Registration_publishes_a_complete_capability();
Duplicate_key_is_refused_and_the_first_stands();
Write_reaches_the_owning_child_through_the_walk();
Stale_revision_is_refused();
Range_type_and_domain_are_enforced();
RequiresReady_follows_the_root_state();
Unknown_key_and_foreign_scope_change_nothing();
Module_invariant_hook_can_refuse();
Units_and_choices_publish_codes_and_labels();

// One-time setup, on the first test to run rather than in a constructor: the
// suite's own Setup return value is itself an assertion below.
METHOD PRIVATE _M_Arm
IF NOT _init THEN
    _init := TRUE;
    _setupOk := _u.Setup(Name := 'Test.CfgUnit');
    _u();
END_IF
END_METHOD

// Walk the real manifest the way a client does — page by page until the key
// appears — so these tests read exactly what the HMI would be given, not an
// internal shortcut into the registry.
METHOD PRIVATE _M_FetchCapability : BOOL
VAR_INPUT
    Key : STRING(160);
END_VAR
VAR
    page  : INT;
    i     : INT;
    pages : INT;
END_VAR
_M_FetchCapability := FALSE;
pages := 1;
FOR page := 0 TO 63 DO
    IF page >= pages THEN
        RETURN;
    END_IF
    _pager.M_Setup(Target := ADR(_page), PageIndex := page, Revision := 1);
    _u.M_AppendConfig(Pager := _pager);
    _pager.M_Finish();
    pages := _page.PageCount;
    FOR i := 1 TO _page.EntryCount DO
        IF _page.Entries[i].WriteKey = Key THEN
            _found := _page.Entries[i];
            _M_FetchCapability := TRUE;
            RETURN;
        END_IF
    END_FOR
END_FOR
END_METHOD

METHOD Registration_publishes_a_complete_capability
TEST('Registration_publishes_a_complete_capability');
_M_Arm();
AssertTrue(Condition := _setupOk,
    Message := 'a registration that fails must fail Setup, not go quiet');
AssertTrue(Condition := _M_FetchCapability(Key := 'probe.settleTime'),
    Message := 'a registered value appears in the root manifest walk');
AssertEquals_STRING(Expected := 'Test.CfgUnit.Child', Actual := _found.Scope,
    Message := 'the capability is scoped to the module that owns it');
AssertTrue(Condition := _found.Writable,
    Message := 'registration is what makes an entry writable (3.10.2)');
AssertEquals_UDINT(Expected := 1, Actual := _found.WriteRevision,
    Message := 'a writable entry carries a non-zero revision');
AssertEquals_DINT(Expected := TO_DINT(E_ConfigValueType.DURATION),
    Actual := TO_DINT(_found.ValueType),
    Message := 'a TIME publishes as DURATION (TC3 3.8)');
AssertEquals_DINT(Expected := TO_DINT(E_ConfigKind.STATION_CFG),
    Actual := TO_DINT(_found.ConfigKind),
    Message := 'deployment data publishes as STATION_CFG');
AssertEquals_STRING(Expected := 'ms', Actual := _found.Unit,
    Message := 'a duration carries its engineering unit');
AssertEquals_STRING(Expected := '500', Actual := _found.ValueText,
    Message := 'the published value is the live target, in whole milliseconds');
AssertTrue(Condition := _found.RequiresReady,
    Message := 'the declared state requirement reaches the client');
AssertEquals_REAL(Expected := 5000.0, Actual := TO_REAL(_found.Maximum),
    Delta := 0.001, Message := 'declared bounds reach the client');
TEST_FINISHED();
END_METHOD

// Core 0.14: a unit is a CODE the HMI translates (the text is derived from it
// for older clients), and a choice names the catalog prefix that labels each of
// its values - so an editor renders a translated dropdown, never a number.
METHOD Units_and_choices_publish_codes_and_labels
TEST('Units_and_choices_publish_codes_and_labels');
_M_Arm();
AssertTrue(Condition := _M_FetchCapability(Key := 'probe.settleTime'),
    Message := 'the duration is published');
AssertEquals_DINT(Expected := TO_DINT(E_EngUnit.MILLISECOND),
    Actual := TO_DINT(_found.UnitCode),
    Message := 'a duration carries the millisecond CODE');
AssertEquals_STRING(Expected := 'ms', Actual := _found.Unit,
    Message := 'and the legacy text is derived from it, not written separately');
AssertTrue(Condition := _M_FetchCapability(Key := 'probe.retries'),
    Message := 'the unitless number is published');
AssertEquals_DINT(Expected := TO_DINT(E_EngUnit.NONE),
    Actual := TO_DINT(_found.UnitCode), Message := 'NONE = no unit');
AssertEquals_STRING(Expected := '', Actual := _found.Unit,
    Message := 'so an HMI shows no unit text');
AssertTrue(Condition := _M_FetchCapability(Key := 'probe.mode'),
    Message := 'the choice is published');
AssertEquals_STRING(Expected := '0|1|2', Actual := _found.EnumDomain,
    Message := 'with its exact accepted values');
AssertEquals_STRING(Expected := 'project.test.modeValue', Actual := _found.EnumLabelKey,
    Message := 'and the catalog prefix that labels each of them');
AssertFalse(Condition := _dup.M_RegisterConfigChoice(Key := 'probe.empty',
    Item := 'StationCfg/Empty', LabelKey := '', Kind := E_ConfigKind.STATION_CFG,
    Storage := E_ConfigStorage.AS_DINT, pTarget := ADR(_dup.Mode), Domain := '',
    EnumLabelKey := '', RequiresReady := FALSE),
    Message := 'a choice with no choices is refused, not accepted as anything');
TEST_FINISHED();
END_METHOD

METHOD Duplicate_key_is_refused_and_the_first_stands
TEST('Duplicate_key_is_refused_and_the_first_stands');
_M_Arm();
AssertTrue(Condition := _dup.Setup(Name := 'Test.CfgDup'),
    Message := 'the probe registers cleanly the first time');
// Re-registering the same key is the §3.10.2 duplicate case. It fails closed,
// which here means the SECOND caller is refused and the first target stays bound
// — nothing can tell which was meant, so the ambiguity is reported, not resolved.
_dupOk := _dup.M_RegisterConfigNumber(Key := 'probe.retries',
    Item := 'StationCfg/Retries2', LabelKey := '', Unit := E_EngUnit.NONE,
    Kind := E_ConfigKind.STATION_CFG, Storage := E_ConfigStorage.AS_DINT,
    pTarget := ADR(_dup.Retries), Minimum := 0.0, Maximum := 99.0,
    RequiresReady := FALSE);
AssertFalse(Condition := _dupOk,
    Message := 'a duplicate (Scope, WriteKey) registration is refused');
// A registration with no target is the other fail-closed case: a capability
// pointing nowhere would publish an editor control that writes into address 0.
AssertFalse(Condition := _dup.M_RegisterConfigFlag(Key := 'probe.nowhere',
        Item := 'StationCfg/Nowhere', LabelKey := '',
        Kind := E_ConfigKind.STATION_CFG, pTarget := 0, RequiresReady := FALSE),
    Message := 'a capability with no target is refused');
TEST_FINISHED();
END_METHOD

METHOD Write_reaches_the_owning_child_through_the_walk
TEST('Write_reaches_the_owning_child_through_the_walk');
_M_Arm();
// The root has no routing code for this key. It finds the owner by Scope.
AssertTrue(Condition := _u.WriteConfig(TargetPath := 'Test.CfgUnit.Child',
        WriteKey := 'probe.retries', Revision := 1, TextValue := '7'),
    Message := 'a valid write is accepted by the owning child');
AssertEquals_DINT(Expected := 7, Actual := _u.Child.Retries,
    Message := 'the child value actually changed');
AssertTrue(Condition := _M_FetchCapability(Key := 'probe.retries'),
    Message := 'the entry is still published after the write');
AssertEquals_STRING(Expected := '7', Actual := _found.ValueText,
    Message := 'the manifest publishes the live value, not a cached copy');
// The root's own registered value goes through the same path.
AssertTrue(Condition := _u.WriteConfig(TargetPath := 'Test.CfgUnit',
        WriteKey := 'probe.cycleLimit', Revision := 1, TextValue := '250'),
    Message := 'the root can own editable values too');
AssertEquals_DINT(Expected := 250, Actual := _u.CycleLimit,
    Message := 'the root value changed');
// A text value with its own revision, proving revision is per capability.
AssertTrue(Condition := _u.WriteConfig(TargetPath := 'Test.CfgUnit.Child',
        WriteKey := 'probe.label', Revision := 2, TextValue := 'line-4'),
    Message := 'a TEXT capability accepts its declared revision');
AssertEquals_STRING(Expected := 'line-4', Actual := _u.Child.Label,
    Message := 'the text value changed');
TEST_FINISHED();
END_METHOD

METHOD Stale_revision_is_refused
TEST('Stale_revision_is_refused');
_M_Arm();
AssertTrue(Condition := _u.WriteConfig(TargetPath := 'Test.CfgUnit.Child',
        WriteKey := 'probe.label', Revision := 2, TextValue := 'keep-me'),
    Message := 'baseline set through the same path under test');
// A client holding an older manifest sends the revision it was given. Accepting
// it would apply a value validated against metadata that no longer exists.
AssertFalse(Condition := _u.WriteConfig(TargetPath := 'Test.CfgUnit.Child',
        WriteKey := 'probe.label', Revision := 1, TextValue := 'stale'),
    Message := 'a revision the capability does not carry is refused');
AssertEquals_STRING(Expected := 'keep-me', Actual := _u.Child.Label,
    Message := 'a refused write changes nothing');
AssertFalse(Condition := _u.WriteConfig(TargetPath := 'Test.CfgUnit.Child',
        WriteKey := 'probe.label', Revision := 0, TextValue := 'stale'),
    Message := 'revision zero is never a valid capability');
AssertEquals_STRING(Expected := 'keep-me', Actual := _u.Child.Label,
    Message := 'still unchanged');
TEST_FINISHED();
END_METHOD

METHOD Range_type_and_domain_are_enforced
TEST('Range_type_and_domain_are_enforced');
_M_Arm();
AssertTrue(Condition := _u.WriteConfig(TargetPath := 'Test.CfgUnit.Child',
        WriteKey := 'probe.retries', Revision := 1, TextValue := '4'),
    Message := 'baseline');
AssertFalse(Condition := _u.WriteConfig(TargetPath := 'Test.CfgUnit.Child',
        WriteKey := 'probe.retries', Revision := 1, TextValue := '11'),
    Message := 'above the declared maximum');
AssertFalse(Condition := _u.WriteConfig(TargetPath := 'Test.CfgUnit.Child',
        WriteKey := 'probe.retries', Revision := 1, TextValue := '-1'),
    Message := 'below the declared minimum');
// The conversion this replaces answers 0 for all three of these, which is why a
// handler built on it accepts garbage as a valid zero (F_TryParseNumber).
AssertFalse(Condition := _u.WriteConfig(TargetPath := 'Test.CfgUnit.Child',
        WriteKey := 'probe.retries', Revision := 1, TextValue := 'abc'),
    Message := 'text that is not a number');
AssertFalse(Condition := _u.WriteConfig(TargetPath := 'Test.CfgUnit.Child',
        WriteKey := 'probe.retries', Revision := 1, TextValue := ''),
    Message := 'empty text');
AssertFalse(Condition := _u.WriteConfig(TargetPath := 'Test.CfgUnit.Child',
        WriteKey := 'probe.retries', Revision := 1, TextValue := '5kg'),
    Message := 'a number with a trailing unit');
AssertFalse(Condition := _u.WriteConfig(TargetPath := 'Test.CfgUnit.Child',
        WriteKey := 'probe.retries', Revision := 1, TextValue := '3.5'),
    Message := 'a fraction into an integer field truncates silently, so it is refused');
AssertEquals_DINT(Expected := 4, Actual := _u.Child.Retries,
    Message := 'six refusals, no change');
// A declared domain is exact: no case folding, no synonyms.
AssertTrue(Condition := _u.WriteConfig(TargetPath := 'Test.CfgUnit.Child',
        WriteKey := 'probe.enabled', Revision := 1, TextValue := 'TRUE'),
    Message := 'baseline');
AssertFalse(Condition := _u.WriteConfig(TargetPath := 'Test.CfgUnit.Child',
        WriteKey := 'probe.enabled', Revision := 1, TextValue := 'yes'),
    Message := 'a value outside the exact enum domain');
AssertTrue(Condition := _u.Child.Enabled, Message := 'flag unchanged');
AssertTrue(Condition := _u.WriteConfig(TargetPath := 'Test.CfgUnit.Child',
        WriteKey := 'probe.enabled', Revision := 1, TextValue := 'FALSE'),
    Message := 'a value inside the domain is accepted');
AssertFalse(Condition := _u.Child.Enabled, Message := 'flag cleared');
TEST_FINISHED();
END_METHOD

METHOD RequiresReady_follows_the_root_state
TEST('RequiresReady_follows_the_root_state');
_M_Arm();
AssertTrue(Condition := _u.WriteConfig(TargetPath := 'Test.CfgUnit.Child',
        WriteKey := 'probe.settleTime', Revision := 1, TextValue := '750'),
    Message := 'accepted while the root is READY');
AssertEquals_TIME(Expected := T#750MS, Actual := _u.Child.SettleTime,
    Message := 'milliseconds land as a duration');
// RequiresReady is a fact about the ROOT, which the child cannot see: the root
// answers it on the way down. Start the Unit and the same write must fail.
AssertTrue(Condition := _u.Start(), Message := 'start');
_u();
AssertFalse(Condition := _u.WriteConfig(TargetPath := 'Test.CfgUnit.Child',
        WriteKey := 'probe.settleTime', Revision := 1, TextValue := '900'),
    Message := 'refused while the root is running');
AssertEquals_TIME(Expected := T#750MS, Actual := _u.Child.SettleTime,
    Message := 'the running machine keeps the value it was judged with');
// A value that did NOT ask for READY is still writable meanwhile.
AssertTrue(Condition := _u.WriteConfig(TargetPath := 'Test.CfgUnit.Child',
        WriteKey := 'probe.retries', Revision := 1, TextValue := '2'),
    Message := 'RequiresReady is per value, not per module');
_u.Stop();
_u();
TEST_FINISHED();
END_METHOD

METHOD Unknown_key_and_foreign_scope_change_nothing
TEST('Unknown_key_and_foreign_scope_change_nothing');
_M_Arm();
AssertTrue(Condition := _u.WriteConfig(TargetPath := 'Test.CfgUnit.Child',
        WriteKey := 'probe.retries', Revision := 1, TextValue := '5'),
    Message := 'baseline');
AssertFalse(Condition := _u.WriteConfig(TargetPath := 'Test.CfgUnit.Child',
        WriteKey := 'probe.notRegistered', Revision := 1, TextValue := '1'),
    Message := 'an unregistered key is refused');
AssertFalse(Condition := _u.WriteConfig(TargetPath := 'Test.CfgUnit.Child',
        WriteKey := '', Revision := 1, TextValue := '1'),
    Message := 'an empty key is refused');
// Right key, wrong owner: the walk asks each module whether the scope is its own,
// so a key that exists elsewhere still finds nobody here.
AssertFalse(Condition := _u.WriteConfig(TargetPath := 'Test.CfgUnit',
        WriteKey := 'probe.retries', Revision := 1, TextValue := '1'),
    Message := 'a child key addressed to the root is refused');
// A path outside this root is rejected before routing even begins (§3.10.2).
AssertFalse(Condition := _u.WriteConfig(TargetPath := 'Other.Unit.Child',
        WriteKey := 'probe.retries', Revision := 1, TextValue := '1'),
    Message := 'a path outside this root is refused');
AssertEquals_DINT(Expected := 5, Actual := _u.Child.Retries,
    Message := 'nothing moved');
TEST_FINISHED();
END_METHOD

METHOD Module_invariant_hook_can_refuse
TEST('Module_invariant_hook_can_refuse');
_M_Arm();
AssertTrue(Condition := _u.WriteConfig(TargetPath := 'Test.CfgUnit.Child',
        WriteKey := 'probe.retries', Revision := 1, TextValue := '6'),
    Message := 'baseline');
_u.M_SetChildRefuse(Text := '9');
// Type-valid, in range, right revision — and still the module's own answer is no.
AssertFalse(Condition := _u.WriteConfig(TargetPath := 'Test.CfgUnit.Child',
        WriteKey := 'probe.retries', Revision := 1, TextValue := '9'),
    Message := 'the owning module may refuse a well-formed candidate');
AssertEquals_UDINT(Expected := 1, Actual := _u.Child.RefusedCount,
    Message := 'the hook ran (the refusal is the module, not the range)');
AssertEquals_DINT(Expected := 6, Actual := _u.Child.Retries,
    Message := 'a hook refusal leaves the value exactly as it was');
_u.M_SetChildRefuse(Text := '');
AssertTrue(Condition := _u.WriteConfig(TargetPath := 'Test.CfgUnit.Child',
        WriteKey := 'probe.retries', Revision := 1, TextValue := '9'),
    Message := 'the same value is accepted once the module stops refusing it');
AssertEquals_DINT(Expected := 9, Actual := _u.Child.Retries,
    Message := 'and now it applied');
TEST_FINISHED();
END_METHOD

END_FUNCTION_BLOCK

// ---- Fraktal_Tests/FB_ProbeConfigPersistence.TcPOU
// §3.8b test double for I_ConfigPersistence. A real durability provider talks
// to the runtime over ADS and completes when it completes, which is not
// something a scan-stepped test can drive; this one is driven explicitly so a
// suite can hold a write PENDING, complete it, or fail it on demand.
//
// It is a TEST fixture and lives in the test project, not in the library: C8
// forbids exactly this shape shipping inside a reusable type (§5.7).
FUNCTION_BLOCK FB_ProbeConfigPersistence IMPLEMENTS I_ConfigPersistence
VAR_OUTPUT
    Requests : UDINT;         // proves the root actually asked, not just published
END_VAR
VAR
    _busy       : BOOL;
    _failed     : BOOL;
    _refuse     : BOOL;       // M_Request itself is refused (a store that will not start)
    _holdBusy   : BOOL;       // stay busy until the test says otherwise
END_VAR

;

METHOD M_Request : BOOL
Requests := Requests + 1;
IF _refuse THEN
    M_Request := FALSE;
    RETURN;
END_IF
_busy := TRUE;
M_Request := TRUE;
END_METHOD

METHOD M_Cyclic : BOOL
IF _busy AND NOT _holdBusy THEN
    _busy := FALSE;                      // completes on the very next scan
END_IF
M_Cyclic := _busy;
END_METHOD

METHOD M_Failed : BOOL
M_Failed := _failed;
END_METHOD

// Keep an accepted write in flight, so a suite can observe PersistPending.
METHOD M_SetHold
VAR_INPUT
    Hold : BOOL;
END_VAR
_holdBusy := Hold;
END_METHOD

// Decide what the NEXT completion reports. Refuse = the store will not even
// start, which §3.8b treats as a failure and not as a quiet no-op.
METHOD M_SetOutcome
VAR_INPUT
    Failed : BOOL;
    Refuse : BOOL;
END_VAR
_failed := Failed;
_refuse := Refuse;
END_METHOD

END_FUNCTION_BLOCK

// ---- Fraktal_Tests/FB_Shift_Tests.TcPOU
// Core §8.5.2 under test. The shift boundary is driven through M_ShiftTick with
// synthetic UTC times - the same method the base calls every scan with the real
// clock - and the units are never cycled, so the real clock cannot interfere.
FUNCTION_BLOCK FB_Shift_Tests EXTENDS TcUnit.FB_TestSuite
VAR
    _u    : FB_ProbeLineUnit;
    _bare : FB_ProbeConfigUnit;
    _init : BOOL;
    _i : INT;
    _day : DT;
    _w1, _w2, _w3, _w4, _w5, _w6 : BOOL;
END_VAR

IF NOT _init THEN
    _init := TRUE;
    _u.Setup(Name := 'Test.Shift', Role := E_LineRole.OWNER, Source := 0,
        StaleAfterMs := 0, ExtraKey := FALSE);
    _u.SetLine(pLine := ADR(_u.Line));
    _bare.Setup(Name := 'Test.NoLine');
    // The calendar is PERSISTENT line data: set it every run.
    _u.WriteConfig(TargetPath := 'Test.Shift', WriteKey := 'line.shift.utcOffsetMin',
        Revision := 1, TextValue := '0');
    _u.WriteConfig(TargetPath := 'Test.Shift', WriteKey := 'line.shift.1.startMin',
        Revision := 1, TextValue := '360');
    _u.WriteConfig(TargetPath := 'Test.Shift', WriteKey := 'line.shift.2.startMin',
        Revision := 1, TextValue := '840');
    _u.WriteConfig(TargetPath := 'Test.Shift', WriteKey := 'line.shift.3.startMin',
        Revision := 1, TextValue := '1320');
    _u.WriteConfig(TargetPath := 'Test.Shift', WriteKey := 'line.shift.4.startMin',
        Revision := 1, TextValue := '-1');
END_IF
Current_shift_follows_the_calendar_and_wraps_midnight();
A_boundary_closes_the_shift_with_its_figures();
An_unsynchronized_boundary_is_recorded_as_such();
A_manual_reset_mid_shift_is_recorded();
The_history_is_bounded_and_newest_first();
No_line_means_no_shift_accounting();

METHOD Current_shift_follows_the_calendar_and_wraps_midnight
TEST('Current_shift_follows_the_calendar_and_wraps_midnight');
IF NOT _w1 THEN
    AssertEquals_INT(Expected := 3, Actual := _u.Line.M_CurrentShift(MinuteOfDay := 300),
        Message := 'before the first start of the day is the LAST shift of the day before');
    AssertEquals_INT(Expected := 1, Actual := _u.Line.M_CurrentShift(MinuteOfDay := 360),
        Message := 'a shift starts at its start minute');
    AssertEquals_INT(Expected := 1, Actual := _u.Line.M_CurrentShift(MinuteOfDay := 839),
        Message := 'and runs until the next used shift');
    AssertEquals_INT(Expected := 2, Actual := _u.Line.M_CurrentShift(MinuteOfDay := 840),
        Message := 'which then takes over');
    AssertEquals_INT(Expected := 3, Actual := _u.Line.M_CurrentShift(MinuteOfDay := 1439),
        Message := 'up to midnight');
    _u.WriteConfig(TargetPath := 'Test.Shift', WriteKey := 'line.shift.utcOffsetMin',
        Revision := 1, TextValue := '120');
    AssertEquals_DINT(Expected := 360, Actual := _u.Line.M_MinuteOfDay(Now := DT#2026-09-27-04:00:00),
        Message := 'the line offset turns the UTC clock into local minutes');
    _u.WriteConfig(TargetPath := 'Test.Shift', WriteKey := 'line.shift.utcOffsetMin',
        Revision := 1, TextValue := '-60');
    AssertEquals_DINT(Expected := 1380, Actual := _u.Line.M_MinuteOfDay(Now := DT#2026-09-27-00:00:00),
        Message := 'a negative offset wraps back across midnight');
    _u.WriteConfig(TargetPath := 'Test.Shift', WriteKey := 'line.shift.utcOffsetMin',
        Revision := 1, TextValue := '0');
    _w1 := TRUE;
END_IF
TEST_FINISHED();
END_METHOD

METHOD A_boundary_closes_the_shift_with_its_figures
TEST('A_boundary_closes_the_shift_with_its_figures');
IF NOT _w2 THEN
    AssertFalse(Condition := _u.M_ShiftTick(Now := DT#2026-09-27-13:00:00, Synchronized := TRUE),
        Message := 'the first evaluation only starts accounting');
    AssertEquals_INT(Expected := 1, Actual := _u.CurrentShift, Message := 'in shift 1');
    _u.CountGood();
    _u.CountGood();
    _u.CountGood();
    AssertFalse(Condition := _u.M_ShiftTick(Now := DT#2026-09-27-13:59:59, Synchronized := TRUE),
        Message := 'no boundary, nothing closes');
    AssertTrue(Condition := _u.M_ShiftTick(Now := DT#2026-09-27-14:00:00, Synchronized := TRUE),
        Message := 'the boundary closes the shift');
    AssertEquals_INT(Expected := 1, Actual := _u.ShiftHistory[1].ShiftIndex, Message := 'the one that ended');
    AssertEquals_UDINT(Expected := 3, Actual := _u.ShiftHistory[1].GoodCount,
        Message := 'with the figures exactly as they stood at the boundary');
    AssertTrue(Condition := _u.ShiftHistory[1].StartAt = DT#2026-09-27-13:00:00, Message := 'from when accounting began');
    AssertTrue(Condition := _u.ShiftHistory[1].EndAt = DT#2026-09-27-14:00:00, Message := 'to the boundary');
    AssertTrue(Condition := _u.ShiftHistory[1].TimeSynchronized, Message := 'on a synchronized clock');
    AssertEquals_UDINT(Expected := 0, Actual := _u.GoodCount, Message := 'and the count starts again');
    AssertEquals_INT(Expected := 2, Actual := _u.CurrentShift, Message := 'for shift 2');
    _w2 := TRUE;
END_IF
TEST_FINISHED();
END_METHOD

METHOD An_unsynchronized_boundary_is_recorded_as_such
TEST('An_unsynchronized_boundary_is_recorded_as_such');
IF NOT _w3 THEN
    AssertTrue(Condition := _u.M_ShiftTick(Now := DT#2026-09-27-22:00:00, Synchronized := FALSE),
        Message := 'a boundary on an unsynchronized clock still closes the shift');
    AssertEquals_INT(Expected := 2, Actual := _u.ShiftHistory[1].ShiftIndex, Message := 'shift 2');
    AssertFalse(Condition := _u.ShiftHistory[1].TimeSynchronized,
        Message := 'and the record says the clock was not to be trusted');
    _w3 := TRUE;
END_IF
TEST_FINISHED();
END_METHOD

METHOD A_manual_reset_mid_shift_is_recorded
TEST('A_manual_reset_mid_shift_is_recorded');
IF NOT _w4 THEN
    AssertTrue(Condition := _u.ResetOee(), Message := 'a hand reset during shift 3');
    AssertTrue(Condition := _u.M_ShiftTick(Now := DT#2026-09-28-06:00:00, Synchronized := TRUE),
        Message := 'the night shift closes the next morning');
    AssertEquals_INT(Expected := 3, Actual := _u.ShiftHistory[1].ShiftIndex, Message := 'shift 3');
    AssertTrue(Condition := _u.ShiftHistory[1].ManualReset,
        Message := 'its total is marked as partial, never silently');
    AssertTrue(Condition := _u.M_ShiftTick(Now := DT#2026-09-28-14:00:00, Synchronized := TRUE),
        Message := 'the next shift closes');
    AssertFalse(Condition := _u.ShiftHistory[1].ManualReset, Message := 'and the mark belonged to one shift only');
    _w4 := TRUE;
END_IF
TEST_FINISHED();
END_METHOD

METHOD The_history_is_bounded_and_newest_first
TEST('The_history_is_bounded_and_newest_first');
IF NOT _w5 THEN
    _day := DT#2026-10-01-00:00:00;
    FOR _i := 1 TO 12 DO
        _u.M_ShiftTick(Now := _day + T#6H, Synchronized := TRUE);
        _u.M_ShiftTick(Now := _day + T#14H, Synchronized := TRUE);
        _day := _day + T#24H;
    END_FOR
    AssertEquals_INT(Expected := 8, Actual := _u.ShiftHistoryCount, Message := 'the history is bounded');
    AssertTrue(Condition := _u.ShiftHistoryTruncated, Message := 'and says it dropped the oldest');
    AssertTrue(Condition := _u.ShiftHistory[1].EndAt = _day - T#24H + T#14H,
        Message := 'newest first');
    _w5 := TRUE;
END_IF
TEST_FINISHED();
END_METHOD

METHOD No_line_means_no_shift_accounting
TEST('No_line_means_no_shift_accounting');
IF NOT _w6 THEN
    AssertFalse(Condition := _bare.M_ShiftTick(Now := DT#2026-09-27-14:00:00, Synchronized := TRUE),
        Message := 'a Unit that references no line closes nothing');
    AssertEquals_INT(Expected := 0, Actual := _bare.CurrentShift, Message := 'and is in no shift');
    _w6 := TRUE;
END_IF
TEST_FINISHED();
END_METHOD

END_FUNCTION_BLOCK

// ---- Fraktal_Tests/FB_ProbeLineUnit.TcPOU
// §3.8e probe root: holds one FB_LineData as a test fixture and registers the
// line's values on it, exactly as a project would. The line is NOT registered as
// a child: the probe only references it (SetLine), as a root on a line does, and
// edits it through its own scope. ExtraKey registers a second line value the
// owner does not have, so a mirror built with it cannot apply the owner's line whole.
FUNCTION_BLOCK FB_ProbeLineUnit EXTENDS FB_UnitBase
VAR_OUTPUT
    Line : FB_LineData;
END_VAR
VAR_INPUT
    Takt  : DINT := 1000;
    Extra : DINT;
END_VAR

Cyclic();

METHOD Setup : BOOL
VAR_INPUT
    Name         : STRING(80);
    Role         : E_LineRole;
    Source       : I_LineSource;
    StaleAfterMs : UDINT;
    ExtraKey     : BOOL;
END_VAR
_M_SetName(Name);
StallTime := T#0S;
Setup := Line.Setup(Name := CONCAT(Name, 'Line'), LineId := 'L1', Role := Role,
    Source := Source, StaleAfterMs := StaleAfterMs);
Setup := Line.M_RegisterConfigNumber(Key := 'line.taktMs', Item := 'LineCfg/TaktMs',
    LabelKey := 'project.test.taktMs', Unit := E_EngUnit.MILLISECOND, Kind := E_ConfigKind.LINE_CFG,
    Storage := E_ConfigStorage.AS_DINT, pTarget := ADR(Takt), Minimum := 0.0,
    Maximum := 100000.0, RequiresReady := FALSE) AND Setup;
IF ExtraKey THEN
    Setup := Line.M_RegisterConfigNumber(Key := 'line.extra', Item := 'LineCfg/Extra',
        LabelKey := 'project.test.extra', Unit := E_EngUnit.NONE, Kind := E_ConfigKind.LINE_CFG,
        Storage := E_ConfigStorage.AS_DINT, pTarget := ADR(Extra), Minimum := 0.0,
        Maximum := 10.0, RequiresReady := FALSE) AND Setup;
END_IF
Setup := SetLine(pLine := ADR(Line)) AND Setup;
END_METHOD

METHOD PROTECTED _M_Dispatch
_M_SetStep(StepNo := 100, StepName := 'project.test.stepA', Awaits := 0,
    AwaitingLabel := '', TimeClass := E_TimeClass.WORK, ExpectedTime := T#0S);
END_METHOD

END_FUNCTION_BLOCK

// ---- Fraktal_Tests/FB_LineData_Tests.TcPOU
// Core §3.8e under test: one owner, read-only mirrors applied whole.
// Every unit runs every scan at the top of the suite, so a mirror polls exactly as
// it would on a station; the tests only observe.
FUNCTION_BLOCK FB_LineData_Tests EXTENDS TcUnit.FB_TestSuite
VAR
    _owner, _mirror, _odd, _flaky, _adsMirror : FB_ProbeLineUnit;
    _src, _oddSrc, _flakySrc : FB_ProbeLineSource;
    _ads : FB_LineAdsSource;
    _init : BOOL;
    _rev : UDINT;
    _takt : DINT;
    _staleSeen : BOOL;
    _n2, _n4, _n5, _n6 : INT;
    _k : INT;
    _found : STRING(80);
    _w1, _w2, _w3, _w4, _w5, _w6, _w7 : BOOL;
    _probe : DINT;
END_VAR

IF NOT _init THEN
    _init := TRUE;
    _owner.Setup(Name := 'Test.LineOwner', Role := E_LineRole.OWNER, Source := 0,
        StaleAfterMs := 0, ExtraKey := FALSE);
    _src.Setup(pOwner := ADR(_owner.Line));
    _oddSrc.Setup(pOwner := ADR(_owner.Line));
    _flakySrc.Setup(pOwner := ADR(_owner.Line));
    _ads.Setup(NetId := '', Port := 851, Symbol := 'PRG_TcUnitRunner.LineTests._owner.Line.Image');
    _mirror.Setup(Name := 'Test.LineMirror', Role := E_LineRole.MIRROR, Source := _src,
        StaleAfterMs := 5000, ExtraKey := FALSE);
    _odd.Setup(Name := 'Test.LineOdd', Role := E_LineRole.MIRROR, Source := _oddSrc,
        StaleAfterMs := 5000, ExtraKey := TRUE);
    _flaky.Setup(Name := 'Test.LineFlaky', Role := E_LineRole.MIRROR, Source := _flakySrc,
        StaleAfterMs := 0, ExtraKey := FALSE);
    _adsMirror.Setup(Name := 'Test.LineAds', Role := E_LineRole.MIRROR, Source := _ads,
        StaleAfterMs := 5000, ExtraKey := FALSE);
END_IF
_owner();
_mirror();
_odd();
_flaky();
_adsMirror();
The_owner_revision_rises_with_every_accepted_write();
A_mirror_applies_the_owner_revision_whole();
A_mirror_refuses_a_direct_write();
A_mirror_that_cannot_apply_a_revision_applies_nothing();
A_mirror_without_updates_goes_stale_and_recovers();
The_ADS_source_reads_the_owner_image();
A_line_is_no_child_and_its_keys_are_its_own();

METHOD The_owner_revision_rises_with_every_accepted_write
TEST('The_owner_revision_rises_with_every_accepted_write');
IF NOT _w1 THEN
    _rev := _owner.Line.OutImm.Revision;
    AssertTrue(Condition := _owner.WriteConfig(TargetPath := 'Test.LineOwner',
        WriteKey := 'line.taktMs', Revision := 1, TextValue := '1200'),
        Message := 'a line value is edited at the owner like any other value');
    _owner();
    AssertEquals_UDINT(Expected := _rev + 1, Actual := _owner.Line.OutImm.Revision,
        Message := 'the accepted write raised the line revision');
    AssertEquals_UDINT(Expected := _rev + 1, Actual := _owner.Line.Image.Revision,
        Message := 'and the whole line was republished at it');
    // Found by key: the line also carries its shift calendar (§8.5.2), registered first.
    _found := '';
    FOR _k := 1 TO _owner.Line.Image.Count DO
        IF _owner.Line.Image.Records[_k].WriteKey = 'line.taktMs' THEN
            _found := _owner.Line.Image.Records[_k].ValueText;
        END_IF
    END_FOR
    AssertEquals_STRING(Expected := '1200', Actual := _found,
        Message := 'carrying the new value');
    _w1 := TRUE;
END_IF
TEST_FINISHED();
END_METHOD

METHOD A_mirror_applies_the_owner_revision_whole
TEST('A_mirror_applies_the_owner_revision_whole');
IF NOT _w2 THEN
    _n2 := _n2 + 1;
    IF (_mirror.Line.OutImm.Revision <> _owner.Line.OutImm.Revision) AND (_n2 < 20) THEN
        RETURN;                           // across scans: a mirror polls its source
    END_IF
    AssertEquals_UDINT(Expected := _owner.Line.OutImm.Revision, Actual := _mirror.Line.OutImm.Revision,
        Message := 'the mirror holds the owner revision');
    AssertEquals_DINT(Expected := _owner.Takt, Actual := _mirror.Takt,
        Message := 'and the owner value, applied through its own typed handler');
    AssertEquals_STRING(Expected := 'Test.LineOwnerLine', Actual := _mirror.Line.OutImm.Owner,
        Message := 'and names the copy it came from');
    _w2 := TRUE;
END_IF
TEST_FINISHED();
END_METHOD

METHOD A_mirror_refuses_a_direct_write
TEST('A_mirror_refuses_a_direct_write');
IF NOT _w3 THEN
    _takt := _mirror.Takt;
    AssertFalse(Condition := _mirror.WriteConfig(TargetPath := 'Test.LineMirror',
        WriteKey := 'line.taktMs', Revision := 1, TextValue := '5'),
        Message := 'two editable copies of one fact are the drift line data removes');
    AssertEquals_DINT(Expected := _takt, Actual := _mirror.Takt, Message := 'nothing changed');
    _w3 := TRUE;
END_IF
TEST_FINISHED();
END_METHOD

METHOD A_mirror_that_cannot_apply_a_revision_applies_nothing
TEST('A_mirror_that_cannot_apply_a_revision_applies_nothing');
IF NOT _w4 THEN
    _n4 := _n4 + 1;
    IF _n4 < 5 THEN
        RETURN;
    END_IF
    AssertEquals_DINT(Expected := 2, Actual := _odd.Line.OutImm.SourceError,
        Message := 'a line with a value the owner does not carry is not applicable whole');
    AssertEquals_DINT(Expected := 1000, Actual := _odd.Takt,
        Message := 'and not even the value both sides share was applied');
    _w4 := TRUE;
END_IF
TEST_FINISHED();
END_METHOD

METHOD A_mirror_without_updates_goes_stale_and_recovers
TEST('A_mirror_without_updates_goes_stale_and_recovers');
IF NOT _w5 THEN
    _n5 := _n5 + 1;
    IF NOT _staleSeen THEN
        _flakySrc.M_SetFail(Fail := TRUE);
        _staleSeen := _flaky.Line.OutImm.Stale;
        IF _n5 < 50 THEN
            RETURN;
        END_IF
    END_IF
    AssertTrue(Condition := _staleSeen, Message := 'a mirror with no update past its window says Stale');
    _flakySrc.M_SetFail(Fail := FALSE);
    IF _flaky.Line.OutImm.Stale AND (_n5 < 100) THEN
        RETURN;
    END_IF
    AssertFalse(Condition := _flaky.Line.OutImm.Stale, Message := 'and recovers by itself');
    AssertEquals_DINT(Expected := 0, Actual := _flaky.Line.OutImm.SourceError,
        Message := 'with no error left standing');
    _w5 := TRUE;
END_IF
TEST_FINISHED();
END_METHOD

METHOD The_ADS_source_reads_the_owner_image
TEST('The_ADS_source_reads_the_owner_image');
IF NOT _w6 THEN
    _n6 := _n6 + 1;
    IF (_adsMirror.Line.OutImm.Revision <> _owner.Line.OutImm.Revision) AND (_n6 < 300) THEN
        RETURN;
    END_IF
    AssertEquals_UDINT(Expected := _owner.Line.OutImm.Revision, Actual := _adsMirror.Line.OutImm.Revision,
        Message := 'a mirror fed over ADS by symbol reaches the owner revision');
    AssertEquals_DINT(Expected := _owner.Takt, Actual := _adsMirror.Takt,
        Message := 'and applies the owner value');
    AssertEquals_DINT(Expected := 0, Actual := _adsMirror.Line.OutImm.SourceError,
        Message := 'with no transport error');
    _w6 := TRUE;
END_IF
TEST_FINISHED();
END_METHOD

METHOD A_line_is_no_child_and_its_keys_are_its_own
TEST('A_line_is_no_child_and_its_keys_are_its_own');
IF NOT _w7 THEN
    // §3.8e(a): the line is referenced, never registered, so it has no path under
    // the root; its values are the root's line data, reached by the root's scope.
    AssertFalse(Condition := _owner.WriteConfig(TargetPath := 'Test.LineOwner.Line',
        WriteKey := 'line.taktMs', Revision := 1, TextValue := '1300'),
        Message := 'a line is not a child of the root that references it');
    // One key space per kind: a line value is keyed line.*, and nothing else is.
    AssertFalse(Condition := _owner.Line.M_RegisterConfigNumber(Key := 'taktMs2',
        Item := 'LineCfg/X', LabelKey := '', Unit := E_EngUnit.NONE,
        Kind := E_ConfigKind.LINE_CFG, Storage := E_ConfigStorage.AS_DINT,
        pTarget := ADR(_probe), Minimum := 0.0, Maximum := 1.0, RequiresReady := FALSE),
        Message := 'a line value without the line. prefix is refused');
    AssertFalse(Condition := _owner.M_RegisterConfigNumber(Key := 'line.stolen',
        Item := 'StationCfg/X', LabelKey := '', Unit := E_EngUnit.NONE,
        Kind := E_ConfigKind.STATION_CFG, Storage := E_ConfigStorage.AS_DINT,
        pTarget := ADR(_probe), Minimum := 0.0, Maximum := 1.0, RequiresReady := FALSE),
        Message := 'and a station value may not take a line key');
    _w7 := TRUE;
END_IF
TEST_FINISHED();
END_METHOD

END_FUNCTION_BLOCK

// ---- Fraktal_Tests/FB_ProbeLineSource.TcPOU
// §3.8e test source: an owner on this controller, with a failure the test can
// switch on. A test seam, so it lives here and never in the library (lint C8).
FUNCTION_BLOCK FB_ProbeLineSource IMPLEMENTS I_LineSource
VAR
    {attribute 'OPC.UA.DA' := '0'}
    _owner : POINTER TO FB_LineData;
    _fail  : BOOL;
END_VAR

;

METHOD Setup : BOOL
VAR_INPUT
    pOwner : POINTER TO FB_LineData;
END_VAR
_owner := pOwner;
Setup := (pOwner <> 0);
END_METHOD

METHOD M_SetFail
VAR_INPUT
    Fail : BOOL;
END_VAR
_fail := Fail;
END_METHOD

METHOD M_Poll : BOOL
VAR_IN_OUT
    Image : ST_LineImage;
END_VAR
M_Poll := FALSE;
IF _fail OR (_owner = 0) THEN
    RETURN;
END_IF
Image := _owner^.Image;
M_Poll := TRUE;
END_METHOD

METHOD M_Error : DINT
M_Error := SEL(_fail, 0, 99);
END_METHOD

END_FUNCTION_BLOCK

// ---- Fraktal_Tests/PRG_TcUnitRunner.TcPOU
// Core §5.7 / TC3 §5.7 — one open-ended gate: every suite joins unchanged (§6.8, H.6)
// Press-example suites (FB_PressDemoUnit_Tests, FB_FaultRecovery_Tests) run
// from Examples/PressDemo/PressTests.plcproj - see that manifest for why.
PROGRAM PRG_TcUnitRunner
VAR
    BaseTests      : FB_Base_Tests;
    PermTests      : FB_PermIntlk_Tests;
    PowerGroupTests: FB_PowerGroupCM_Tests;
    TwoHandTests   : FB_TwoHandStartCM_Tests;
    TimingTests    : FB_Timing_Tests;
    UnitTests      : FB_Unit_Tests;
    ConnectorTests : FB_Connector_Tests;
    CylinderTests  : FB_CylinderCM_Tests;
    DecisionTests  : FB_Decision_Tests;
    ConfigurableCylinderTests : FB_ConfigurableCylinderCM_Tests;
    ClampTests     : FB_ClampEM_Tests;
    UnitTierTests : FB_UnitTier_Tests;
    HmiTests       : FB_Hmi_Tests;
    HostEventTests : FB_HostEvent_Tests;
    IoTopologyTests: FB_IoTopologyPublisher_Tests;
    InputModuleTests: FB_InputCM_Tests;
    AccessTests    : FB_Access_Tests;
    AlarmLogTests  : FB_AlarmLog_Tests;
    ManualCmdTests : FB_ManualCmd_Tests;
    MultiRootTests : FB_MultiRoot_Tests;
    OeeTests       : FB_Oee_Tests;
    ReleaseTests   : FB_Release_Tests;
    ShelveTests    : FB_Shelve_Tests;
    TcpDeviceTests : FB_TcpDev_Tests;
    PartTraceTests : FB_PartTrace_Tests;
    SystemInfrastructureTests : FB_SystemInfrastructure_Tests;
    SequenceRaiseTests : FB_SequenceRaise_Tests;
    SequenceParTests : FB_SequencePar_Tests;
    StateFlagTests : FB_StateFlag_Tests;
    AxisTests : FB_Axis_Tests;
    RobotPlannerTests : FB_RobotPlanner_Tests;
    RobotConnectorTests : FB_RobotConnector_Tests;
    RobotCmTests : FB_RobotCM_Tests;
    AxisJogTests : FB_AxisJog_Tests;
    SeparatorTests : FB_Separator_Tests;
    EngineeringTests : FB_Engineering_Tests;
    ConfigWriteTests : FB_ConfigWrite_Tests;
    ConfigDurabilityTests : FB_ConfigDurability_Tests;
    ConfigSetTests : FB_ConfigSet_Tests;
    DataClassTests : FB_DataClass_Tests;
    ModelDataTests : FB_ModelData_Tests;
    Sha256Tests : FB_Sha256_Tests;
    LineTests : FB_LineData_Tests;
    ShiftTests : FB_Shift_Tests;
    HandoverTests : FB_Handover_Tests;
    AccessPersistenceTests : FB_AccessPersistence_Tests;
    PlatformHealthTests : FB_PlatformHealth_Tests;
    PersistMediumTests : FB_PersistMedium_Tests;
    LiveConfigTests : FB_LiveConfig_Tests;
END_VAR

TcUnit.RUN();
// Not a suite: the live target-provider harness for isolated acceptance.
PRG_PlatformAcceptance();

END_PROGRAM

// ---- Fraktal_Tests/FB_Timing_Tests.TcPOU
// Core §8.11.4 under test: exact aggregate math, classified profiler publication,
// and the base class capturing a tagged command's row — proven ONCE for all types.
FUNCTION_BLOCK FB_Timing_Tests EXTENDS TcUnit.FB_TestSuite
VAR
    _row : ST_TimingRow;
    _pf  : FB_CycleProfiler;
    _p   : FB_ProbeCM;
    _wp  : BOOL;
    _profilerPhase : INT;
END_VAR

TimingUpdate_math_is_exact();
Profiler_publishes_classified_cycle();
Base_captures_tagged_command_row();

METHOD TimingUpdate_math_is_exact
TEST('TimingUpdate_math_is_exact');
F_TimingUpdate(Row := _row, DurMs := 100);
F_TimingUpdate(Row := _row, DurMs := 200);
F_TimingUpdate(Row := _row, DurMs := 300);
AssertEquals_UDINT(Expected := 3, Actual := _row.Count, Message := 'count');
AssertEquals_TIME(Expected := T#300MS, Actual := _row.Last, Message := 'last');
AssertEquals_TIME(Expected := T#100MS, Actual := _row.Minimum, Message := 'minimum');
AssertEquals_TIME(Expected := T#300MS, Actual := _row.Maximum, Message := 'maximum');
AssertEquals_TIME(Expected := T#200MS, Actual := _row.Avg,  Message := 'running mean 100,200,300 -> 200');
TEST_FINISHED();
END_METHOD

METHOD Profiler_publishes_classified_cycle
TEST('Profiler_publishes_classified_cycle');
// TIME() has millisecond resolution. Keep each cycle open across a real task scan so
// the throughput assertion measures elapsed time instead of inventing a minimum.
CASE _profilerPhase OF
    0:
        _pf.ResetStats();
        // cycle 1: an upstream wait, then work
        _pf.StepChanged(StepNo := 90,  StepName := 'Await pallet', TimeClass := E_TimeClass.WAIT_UPSTREAM, Expected := T#0S);
        _pf.StepChanged(StepNo := 90,  StepName := 'Await pallet', TimeClass := E_TimeClass.WAIT_UPSTREAM, Expected := T#0S);  // refresh: no new entry
        _pf.StepChanged(StepNo := 100, StepName := 'Separate', TimeClass := E_TimeClass.WORK, Expected := T#2S);
        _pf.StepChanged(StepNo := 200, StepName := 'Clamp', TimeClass := E_TimeClass.WORK, Expected := T#0S);
        _profilerPhase := 1;

    1:
        _pf.CycleComplete();
        AssertEquals_TIME(Expected := T#2S, Actual := _pf.LastCycle.Steps[2].Expected,
                          Message  := 'declared guard published for guard-vs-actual (8.11.4c)');
        AssertEquals_INT(Expected := 3, Actual := _pf.LastCycle.NSteps, Message := 'three steps in the waterfall');
        AssertEquals_DINT(Expected := TO_DINT(E_TimeClass.WAIT_UPSTREAM),
                          Actual   := TO_DINT(_pf.LastCycle.Steps[1].TimeClass),
                          Message  := 'wait step carries its declared class (8.11.4f)');
        AssertEquals_DINT(Expected := TO_DINT(E_TimeClass.WORK),
                          Actual   := TO_DINT(_pf.LastCycle.Steps[2].TimeClass),
                          Message  := 'undeclared step defaults to WORK');
        AssertEquals_TIME(Expected := _pf.LastCycle.Total,
                          Actual   := _pf.LastCycle.WorkTime + _pf.LastCycle.WaitTime,
                          Message  := 'Total = WorkTime (real cycle time) + WaitTime');
        AssertEquals_UDINT(Expected := 1, Actual := _pf.LastCycle.CycleNo, Message := 'cycle counter');
        // cycle 2 — aggregates accumulate per StepNo and keep the class
        _pf.StepChanged(StepNo := 90,  StepName := 'Await pallet', TimeClass := E_TimeClass.WAIT_UPSTREAM, Expected := T#0S);
        _pf.StepChanged(StepNo := 100, StepName := 'Separate', TimeClass := E_TimeClass.WORK, Expected := T#0S);
        _pf.StepChanged(StepNo := 200, StepName := 'Clamp', TimeClass := E_TimeClass.WORK, Expected := T#0S);
        _profilerPhase := 2;

    2:
        _pf.CycleComplete();
        AssertEquals_UDINT(Expected := 2, Actual := _pf.LastCycle.CycleNo, Message := 'second cycle published');
        // §8.11.1/§8.11.4 — throughput markers + trend ring follow completed cycles
        AssertEquals_TIME(Expected := _pf.LastCycle.Total, Actual := _pf.LastCycleTime,
                          Message := 'LastCycleTime tracks the completed cycle (8.11.1)');
        AssertTrue(Condition := (_pf.MinCycleTime > T#0S) AND (_pf.MinCycleTime <= _pf.LastCycleTime),
                   Message := 'MinCycleTime is the rolling best (8.11.1)');
        AssertEquals_INT(Expected := 2, Actual := _pf.HistoryHead, Message := 'trend ring advanced per cycle');
        AssertEquals_UDINT(Expected := 2, Actual := _pf.History[2].CycleNo, Message := 'ring carries the cycle number');
        AssertEquals_TIME(Expected := _pf.History[2].WorkTime + _pf.History[2].WaitTime,
                          Actual   := _pf.History[2].Total,
                          Message  := 'ring split reconciles (8.11.4f)');
        AssertEquals_UDINT(Expected := 2, Actual := _pf.StepStats[1].Count, Message := 'per-step aggregate counts cycles');
        AssertEquals_DINT(Expected := 90, Actual := _pf.StepStats[1].Id, Message := 'aggregate keyed by StepNo');
        AssertEquals_DINT(Expected := TO_DINT(E_TimeClass.WAIT_UPSTREAM),
                          Actual   := TO_DINT(_pf.StepStats[1].TimeClass),
                          Message  := 'aggregate row keeps the time class');
        _profilerPhase := 3;
        TEST_FINISHED();
ELSE
    // completed — TcUnit keeps invoking the suite FB while other tests finish
END_CASE
END_METHOD

METHOD Base_captures_tagged_command_row
TEST('Base_captures_tagged_command_row');
IF NOT _wp THEN
    _p.Setup('Test.TimingProbe');
    _wp := TRUE;
END_IF
_p.Execute := TRUE;
_p();
_p.SimDone := TRUE;
_p();                                    // BUSY -> DONE: the base closes the timing row
AssertTrue(Condition := _p.Done, Message := 'probe completed');
AssertEquals_UDINT(Expected := 1, Actual := _p.Timing.Rows[1].Count,
                   Message := 'one completed command recorded (Core 8.11.4a)');
AssertEquals_DINT(Expected := 1, Actual := _p.Timing.Rows[1].Id, Message := 'row keyed by tagged id');
AssertEquals_STRING(Expected := 'PROBE', Actual := _p.Timing.Rows[1].Label,
                    Message := 'row carries the tagged label for the HMI table');
_p.Execute := FALSE;
_p.SimDone := FALSE;
_p();
TEST_FINISHED();
END_METHOD

END_FUNCTION_BLOCK

// ---- Fraktal_Tests/FB_Unit_Tests.TcPOU
// FB_UnitBase suite: mode rejection, run-as-command, stall key, wait-class
// derived Starved, cycle publication, mode change = immediate software abort by default.
FUNCTION_BLOCK FB_Unit_Tests EXTENDS TcUnit.FB_TestSuite
VAR
    _u : FB_ProbeUnit;
    // The config-capability test needs a Unit that is READY. _u is not: the
    // stall test starts it and FB_ProbeUnit only reaches its _M_EndOfCycle stop
    // point when SimB is set, so a Stop() is never granted and it stays BUSY.
    // A shared fixture in a non-shareable state is what that test was really
    // measuring; give it its own.
    _uCfg : FB_ProbeUnit;
    _w : BOOL;
    _wCfg : BOOL;
    _pager : FB_ConfigPager;
    _page : ST_ConfigPage;
END_VAR

Unit_run_stall_classes_and_cycle();
Unit_mode_change_is_estop_by_default();
Sequence_rows_belong_to_the_active_mode();
Unit_config_capability_is_typed_and_fail_closed();

METHOD Unit_run_stall_classes_and_cycle
TEST('Unit_run_stall_classes_and_cycle');
IF NOT _w THEN
    _u.Setup('Test.Unit');
    _w := TRUE;
END_IF
AssertFalse(Condition := _u.SetMode(Mode := E_Mode.CALIBRATION),
            Message := 'unsupported mode rejected gracefully (3.4/3.7)');
AssertTrue(Condition := _u.Start(), Message := 'Start issues the run command (6 intro)');
_u();                                         // edge -> BUSY, step 100 set
_u();                                         // stall guard (T#0S) fires -> pending
AssertTrue(Condition := _u.Busy, Message := 'running');
AssertEquals_DWORD(Expected := TO_DWORD(E_Reason.STEP_STALLED),
                   Actual   := TO_DWORD(_u.Pending.ReasonCode),
                   Message  := 'stall is a PENDING reason, not a fault (6.9)');
AssertEquals_STRING(Expected := 'std.diagnostic.stepStalled',
                    Actual   := _u.Pending.Description,
                    Message  := 'stall publishes a stable key; CurrentStep carries context');
AssertFalse(Condition := _u.Error, Message := 'no fault from a stall');
_u.SimA := TRUE;
_u();                                         // -> step 200 (WAIT_UPSTREAM)
_u();
AssertTrue(Condition := _u.Starved,
           Message := 'Starved derived from the step wait class (8.11.4f/8.11.3)');
_u.Stop();
_u.SimB := TRUE;
_u();                                         // -> step 30
_u();                                         // EndOfCycle: publish + complete + release
_u();                                         // reset -> READY
AssertFalse(Condition := _u.Busy, Message := 'stopped after cycle (3.3)');
AssertEquals_INT(Expected := 2, Actual := _u.Profiler.LastCycle.NSteps,
                 Message := 'cycle profile published with both steps (8.11.4b)');
TEST_FINISHED();
END_METHOD

METHOD Unit_config_capability_is_typed_and_fail_closed
VAR
    i : INT;
    found : BOOL;
    pageIndex : INT;
    pageCount : INT;
END_VAR
TEST('Unit_config_capability_is_typed_and_fail_closed');
// Latched like the stall test above it. Without this the method re-ran every
// scan against a Unit that test leaves BUSY, and the READY-gated write below
// was then refused CORRECTLY - so the failure measured the mode gate rather
// than the capability it names.
IF NOT _wCfg THEN
_wCfg := TRUE;
// Never started, so it is READY - which is what RequiresReady asks for.
AssertTrue(Condition := _uCfg.Setup('Test.Unit'),
    Message := 'the config fixture sets up under the owning path');
_uCfg();
AssertFalse(Condition := _uCfg.Busy,
    Message := 'the Unit is idle before a READY-gated write is attempted');
found := FALSE;
_pager.M_Setup(Target := ADR(_page), PageIndex := 0, Revision := 1);
_uCfg.M_AppendConfig(Pager := _pager);
_pager.M_Finish();
pageCount := _page.PageCount;
// The manifest is a bounded window. Search every advertised page instead of
// coupling this contract test to the current number/order of base entries.
FOR pageIndex := 0 TO pageCount - 1 DO
    _pager.M_Setup(Target := ADR(_page), PageIndex := pageIndex, Revision := 1);
    _uCfg.M_AppendConfig(Pager := _pager);
    _pager.M_Finish();
    FOR i := 1 TO _page.EntryCount DO
        IF _page.Entries[i].WriteKey = 'unit.modePolicy.3.shield' THEN
            found := TRUE;
            AssertTrue(Condition := _page.Entries[i].Writable,
                Message := 'mode policy is an explicit write capability');
            AssertEquals_UDINT(Expected := 1, Actual := _page.Entries[i].WriteRevision,
                Message := 'write capability has a non-zero schema revision');
            AssertTrue(Condition := _page.Entries[i].RequiresReady,
                Message := 'capability publishes its READY-state constraint');
        END_IF
    END_FOR
END_FOR
AssertTrue(Condition := found, Message := 'stable mode-policy key is manifest-served');
AssertTrue(Condition := _uCfg.WriteConfig(TargetPath := 'Test.Unit',
    WriteKey := 'unit.modePolicy.3.shield', Revision := 1, TextValue := '0'),
    Message := 'registered exact enum value is accepted while READY');
AssertEquals_DINT(Expected := TO_DINT(E_ModeSwitchShield.INTERRUPTIBLE),
    Actual := TO_DINT(_uCfg.ModePolicy[3].Shield), Message := 'typed handler applied value');
AssertFalse(Condition := _uCfg.WriteConfig(TargetPath := 'Test.Unit',
    WriteKey := 'unit.modePolicy.3.shield', Revision := 2, TextValue := '1'),
    Message := 'stale capability revision is rejected');
AssertFalse(Condition := _uCfg.WriteConfig(TargetPath := 'Test.Unit',
    WriteKey := 'unit.modePolicy.3.shield', Revision := 1, TextValue := '9'),
    Message := 'out-of-domain value is rejected');
AssertFalse(Condition := _uCfg.WriteConfig(TargetPath := 'Other.Unit',
    WriteKey := 'unit.modePolicy.3.shield', Revision := 1, TextValue := '1'),
    Message := 'foreign owner path is rejected');
END_IF
TEST_FINISHED();
END_METHOD

METHOD Sequence_rows_belong_to_the_active_mode
TEST('Sequence_rows_belong_to_the_active_mode');
// The previous test left the Unit in MANUAL having run two AUTO steps, so the §3.13
// table had rows in it when the mode committed. Discovery has no end of its own:
// without a boundary the chart becomes the union of every chain run since boot.
AssertEquals_INT(Expected := 0, Actual := _u.SequenceStepCount,
    Message := 'committing a mode drops the previous mode chain rows');
AssertEquals_INT(Expected := 0, Actual := _u.SequenceStepDef[1].StepNo,
    Message := 'and clears them, so a later row cannot inherit stale text');
// the new mode fills its own table from scratch
AssertTrue(Condition := _u.SetMode(Mode := E_Mode.AUTO), Message := 'back to AUTO');
_u();
_u();
_u();
AssertTrue(Condition := _u.Start(), Message := 'run the AUTO chain again');
_u();
AssertEquals_INT(Expected := 1, Actual := _u.SequenceStepCount,
    Message := 'the chart rebuilds from the mode that is actually running');
TEST_FINISHED();
END_METHOD

METHOD Unit_mode_change_is_estop_by_default
TEST('Unit_mode_change_is_estop_by_default');
_u.SimA := FALSE;
_u.SimB := FALSE;
AssertTrue(Condition := _u.Start(), Message := 're-start');
_u();
AssertTrue(Condition := _u.Busy, Message := 'running again');
AssertTrue(Condition := _u.SetMode(Mode := E_Mode.MANUAL), Message := 'mode request accepted (pending)');
_u();                                         // OnModeExit=0 -> OnAbort (non-safety software abort, 3.14.4)
_u();                                         // release run command, reset
_u();                                         // commit mode
AssertFalse(Condition := _u.Busy, Message := 'chain cancelled by the mode change');
AssertEquals_UDINT(Expected := 1, Actual := _u.ModeExitCount,
    Message := 'OnModeExit runs once for this immediate transition');
AssertEquals_UDINT(Expected := 1, Actual := _u.ModeExitFirstCount,
    Message := 'OnModeExit receives FirstCall exactly once');
AssertEquals_DINT(Expected := TO_DINT(E_Mode.MANUAL),
    Actual := TO_DINT(_u.LastRequestedMode),
    Message := 'OnModeExit receives the pending target mode');
AssertEquals_UDINT(Expected := 1, Actual := _u.ModeChangedCount,
    Message := 'OnModeChanged runs once after commit');
AssertEquals_DINT(Expected := TO_DINT(E_Mode.AUTO),
    Actual := TO_DINT(_u.LastOldMode),
    Message := 'OnModeChanged receives the mode being left');
AssertEquals_DINT(Expected := TO_DINT(E_Mode.MANUAL),
    Actual := TO_DINT(_u.LastNewMode),
    Message := 'OnModeChanged receives the committed mode');
AssertEquals_DINT(Expected := TO_DINT(E_Mode.MANUAL),
                  Actual   := TO_DINT(_u.ModeActive),
                  Message  := 'mode committed after leaving BUSY (3.14.4)');
AssertEquals_DINT(Expected := TO_DINT(E_HostEventKind.MODE_CHANGED),
    Actual := TO_DINT(_u.HostEvents.Ring[_u.HostEvents.RingHead].Kind),
    Message := 'base emits the fixed mode host event once committed');
AssertEquals_STRING(Expected := 'Test.Unit',
    Actual := _u.HostEvents.Ring[_u.HostEvents.RingHead].StationPath,
    Message := 'host event owns the qualified root path');
AssertEquals_STRING(Expected := '1',
    Actual := _u.HostEvents.Ring[_u.HostEvents.RingHead].Value,
    Message := 'new mode is projected in the compact event value');
TEST_FINISHED();
END_METHOD

END_FUNCTION_BLOCK

// ---- Fraktal_Tests/FB_Shelve_Tests.TcPOU
// Core §8.10: shelving suppresses ANNUNCIATION only. Unrationalized -> refuse;
// SAFETY -> refuse; a shelved MANUAL_RESET alarm STILL BLOCKS (the O7 test).
// Auto-expiry timing is runtime-verified (F_Now-driven).
FUNCTION_BLOCK FB_Shelve_Tests EXTENDS TcUnit.FB_TestSuite
VAR
    _log : FB_AlarmLog;
    _s1, _s2, _s3, _s4 : INT;
    _w : BOOL;
END_VAR

IF NOT _w THEN
    _log.RegisterMeta(Reason := 100, OperatorAction := 'act', Consequence := 'cons', Shelvable := TRUE);
    _s1 := _log.Raise(Reason := 100, Text := 'shelvable blocking',
        Source := 'T', Severity := E_Severity.HIGH, Category := E_Category.PROCESS,
        ResetClass := E_ResetClass.MANUAL_RESET);
    _s2 := _log.Raise(Reason := 200, Text := 'no meta',
        Source := 'T', Severity := E_Severity.LOW, Category := E_Category.PROCESS,
        ResetClass := E_ResetClass.AUTO_RESET);
    _s3 := _log.Raise(Reason := 300, Text := 'safety',
        Source := 'T', Severity := E_Severity.HIGH, Category := E_Category.SAFETY,
        ResetClass := E_ResetClass.MANUAL_RESET);
    _s4 := _log.Raise(Reason := E_Reason.TASK_JITTER_HIGH, Text := 'generated',
        Source := 'T', Severity := E_Severity.HIGH, Category := E_Category.PROCESS,
        ResetClass := E_ResetClass.AUTO_RESET);
    _w := TRUE;
END_IF
Unrationalized_refused();
Safety_refused();
Zero_duration_refused();
Shelved_still_blocks();
Generated_metadata_is_authoritative();
Reused_slot_clears_shelf_state();

METHOD Unrationalized_refused
TEST('Unrationalized_refused');
AssertFalse(Condition := _log.Shelve(Slot := _s2, DurationS := 60),
            Message := 'no rationalization record -> not shelvable (§8.10)');
TEST_FINISHED();
END_METHOD

METHOD Generated_metadata_is_authoritative
TEST('Generated_metadata_is_authoritative');
AssertEquals_DINT(Expected := TO_DINT(E_Severity.LOW),
    Actual := TO_DINT(_log.Active[_s4].Severity),
    Message := 'generated priority replaces caller reclassification');
AssertEquals_DINT(Expected := TO_DINT(E_Category.SYSTEM),
    Actual := TO_DINT(_log.Active[_s4].Category),
    Message := 'generated class replaces caller reclassification');
AssertTrue(Condition := _log.Shelve(Slot := _s4, DurationS := 60),
    Message := 'generated shelvability needs no project registration');
AssertFalse(Condition := _log.RegisterMeta(Reason := E_Reason.TASK_JITTER_HIGH,
    OperatorAction := 'override', Consequence := 'override', Shelvable := FALSE),
    Message := 'standard metadata cannot be overridden per project');
AssertFalse(Condition := _log.RegisterMetaFull(Reason := 400,
    OperatorAction := 'act', Consequence := '', Priority := E_Severity.LOW,
    Category := E_Category.PROCESS, Shelvable := FALSE),
    Message := 'external metadata requires a complete consequence');
AssertFalse(Condition := _log.RegisterMetaFull(Reason := 401,
    OperatorAction := 'act', Consequence := 'cons', Priority := 99,
    Category := E_Category.PROCESS, Shelvable := FALSE),
    Message := 'external priority ordinal is bounds checked');
AssertFalse(Condition := _log.RegisterMetaFull(Reason := 402,
    OperatorAction := 'act', Consequence := 'cons', Priority := E_Severity.HIGH,
    Category := E_Category.SAFETY, Shelvable := TRUE),
    Message := 'external Safety metadata cannot enable shelving');
_log.Unshelve(Slot := _s4);
_log.Gone(Slot := _s4);
TEST_FINISHED();
END_METHOD

METHOD Zero_duration_refused
TEST('Zero_duration_refused');
AssertFalse(Condition := _log.Shelve(Slot := _s1, DurationS := 0),
            Message := 'zero-duration shelf cannot become permanent (8.10)');
TEST_FINISHED();
END_METHOD

METHOD Safety_refused
TEST('Safety_refused');
_log.RegisterMeta(Reason := 300, OperatorAction := 'x', Consequence := 'y', Shelvable := TRUE);
AssertFalse(Condition := _log.Shelve(Slot := _s3, DurationS := 60),
            Message := 'SAFETY category never shelvable, even flagged (§8.10)');
TEST_FINISHED();
END_METHOD

METHOD Reused_slot_clears_shelf_state
VAR
    slot : INT;
END_VAR
TEST('Reused_slot_clears_shelf_state');
AssertTrue(Condition := _log.Shelve(Slot := _s1, DurationS := 60), Message := 'shelf before close');
_log.Gone(Slot := _s1);
_log.OperatorReset();
slot := _log.Raise(Reason := 100, Text := 'reused slot',
    Source := 'T', Severity := E_Severity.LOW, Category := E_Category.PROCESS,
    ResetClass := E_ResetClass.AUTO_RESET);
AssertFalse(Condition := _log.Active[slot].Shelved,
            Message := 'new event never inherits a prior occupant shelf');
_log.Gone(Slot := slot);
TEST_FINISHED();
END_METHOD

METHOD Shelved_still_blocks
TEST('Shelved_still_blocks');
AssertTrue(Condition := _log.Blocking, Message := 'MANUAL_RESET alarm blocks before shelve');
AssertTrue(Condition := _log.Shelve(Slot := _s1, DurationS := 60), Message := 'rationalized+flagged shelves OK');
AssertTrue(Condition := _log.Active[_s1].Shelved, Message := 'annunciation suppressed');
AssertTrue(Condition := _log.Blocking, Message := 'STILL BLOCKING while shelved - control untouched (O7)');
AssertTrue(Condition := _log.Unshelve(Slot := _s1), Message := 'unshelve restores');
AssertFalse(Condition := _log.Active[_s1].Shelved, Message := 'flag cleared');
TEST_FINISHED();
END_METHOD

END_FUNCTION_BLOCK

// ---- Fraktal_Tests/FB_SystemInfrastructure_Tests.TcPOU
// Core §2.7/§8.12/§8.13 fault-injection and truth-table coverage.
FUNCTION_BLOCK FB_SystemInfrastructure_Tests EXTENDS TcUnit.FB_TestSuite
VAR
    _log : FB_AlarmLog;
    _stampLog : FB_AlarmLog;
    _health : FB_SystemHealthPublisher;
    _input : ST_SystemHealthInput;
    _healthCfg : ST_SystemHealthParCfg;
    _tower : FB_SignalTower;
    _towerCfg : ST_SignalTowerParCfg;
    _setup : BOOL;
    _slot : INT;
    _towerPhase : INT;
    _towerStarted : TIME;
    _windowsClock : FB_TcWindowsTime;
    _clockSample : ST_TcWindowsClockSampleV1;
    _clockApplied : BOOL;
    _fileClock : FB_TcWindowsTime;
    _fileOps : FB_ProbeFileOps;
    _fileSample : ST_TcWindowsClockSampleV1;
    _fileStep : INT;
    _fileGuard : TON;
    _fileLog : FB_AlarmLog;
END_VAR
VAR CONSTANT
    // Test-runtime only: the observer path is absolute by design (PATH_GENERIC).
    CLOCK_TEST_DIR  : STRING(80) := 'C:\ProgramData\Fraktal\TcUnit';
    CLOCK_TEST_FILE : STRING(80) := 'C:\ProgramData\Fraktal\TcUnit\clock.bin';
END_VAR

Health_fault_edges_are_auto_reset_and_time_qualified();
Tower_mapping_and_bounded_test();
Windows_clock_quality_rejects_bad_and_stale_samples();
Crc32_matches_the_standard_and_the_native_observer();
Windows_clock_file_reader_reads_rejects_and_expires();

METHOD Health_fault_edges_are_auto_reset_and_time_qualified
TEST('Health_fault_edges_are_auto_reset_and_time_qualified');
IF NOT _setup THEN
    _health.Setup(SourcePath := 'Test.Unit.SystemHealth', pAlarmLog := ADR(_log));
    _healthCfg.MaxTaskCycleUs := 2000;
    _healthCfg.MaxTaskJitterUs := 500;
    _setup := TRUE;
END_IF
_input.TaskAvailable := TRUE;
_input.TaskCycleUs := 1000;
_input.TaskJitterUs := 10;
_input.ControllerAvailable := TRUE;
_input.CpuLoadPct := 20.0;
_input.MemoryAvailableMb := 1024;
_input.TimeQuality.Available := TRUE;
_input.TimeQuality.Synchronized := TRUE;
_input.TimeQuality.Source := 'TEST';
_health.Cyclic(Input := _input, ParCfg := _healthCfg, Configured := TRUE);
AssertTrue(Condition := _health.Status.Healthy, Message := 'healthy sample stays healthy');

_input.TimeQuality.Synchronized := FALSE;
_health.Cyclic(Input := _input, ParCfg := _healthCfg, Configured := TRUE);
AssertFalse(Condition := _health.Status.Healthy, Message := 'sync loss degrades health');
AssertEquals_INT(Expected := 1, Actual := _log.NActive, Message := 'one time-sync event opens');
AssertEquals_DWORD(Expected := TO_DWORD(E_Reason.TIME_SYNC_LOST),
    Actual := TO_DWORD(_log.Active[1].ReasonCode), Message := 'registered time-sync reason');

_input.TimeQuality.Synchronized := TRUE;
_health.Cyclic(Input := _input, ParCfg := _healthCfg, Configured := TRUE);
AssertEquals_INT(Expected := 0, Actual := _log.NActive, Message := 'restored sync auto-closes');
AssertEquals_DWORD(Expected := TO_DWORD(E_Reason.TIME_SYNC_LOST),
    Actual := TO_DWORD(_log.Ring[_log.RingHead].ReasonCode), Message := 'closed edge retained');

GVL_FraktalTime.Current.Available := TRUE;
GVL_FraktalTime.Current.Synchronized := FALSE;
_slot := _stampLog.Raise(Reason := E_Reason.NONE, Text := 'test.unsynchronized',
    Source := 'Test.Unit', Severity := E_Severity.LOW,
    Category := E_Category.SYSTEM, ResetClass := E_ResetClass.AUTO_RESET);
AssertFalse(Condition := _stampLog.Active[_slot].ComeTimeSynchronized,
    Message := 'generated timestamp carries unsynchronized quality');
_stampLog.Gone(Slot := _slot);
GVL_FraktalTime.Current.Synchronized := TRUE;
TEST_FINISHED();
END_METHOD

METHOD Tower_mapping_and_bounded_test
TEST('Tower_mapping_and_bounded_test');
CASE _towerPhase OF
    0:
        _tower.Cyclic(MachineState := E_MachineState.PRODUCING,
            AlarmActive := FALSE, HighestSeverity := E_Severity.LOW,
            OperatorActionRequired := FALSE, LampTestRequest := FALSE,
            ParCfg := _towerCfg);
        AssertTrue(Condition := _tower.Status.Green, Message := 'producing maps green');
        _tower.Cyclic(MachineState := E_MachineState.PRODUCING,
            AlarmActive := TRUE, HighestSeverity := E_Severity.HIGH,
            OperatorActionRequired := FALSE, LampTestRequest := FALSE,
            ParCfg := _towerCfg);
        AssertTrue(Condition := _tower.Status.Red AND _tower.Status.Horn
            AND NOT _tower.Status.Green, Message := 'high alarm overrides to red and horn');
        _tower.Cyclic(MachineState := E_MachineState.STOPPED,
            AlarmActive := FALSE, HighestSeverity := E_Severity.LOW,
            OperatorActionRequired := TRUE, LampTestRequest := FALSE,
            ParCfg := _towerCfg);
        AssertTrue(Condition := _tower.Status.Blue, Message := 'operator action maps blue');
        _towerCfg.LampTestDuration := T#2MS;
        _tower.Cyclic(MachineState := E_MachineState.STOPPED,
            AlarmActive := FALSE, HighestSeverity := E_Severity.LOW,
            OperatorActionRequired := FALSE, LampTestRequest := TRUE,
            ParCfg := _towerCfg);
        AssertTrue(Condition := _tower.Status.TestActive AND _tower.Status.Red
            AND _tower.Status.Amber AND _tower.Status.Green AND _tower.Status.Blue
            AND _tower.Status.White AND _tower.Status.Horn,
            Message := 'lamp test drives every semantic output');
        _towerStarted := TIME();
        _towerPhase := 1;
    1:
        _tower.Cyclic(MachineState := E_MachineState.STOPPED,
            AlarmActive := FALSE, HighestSeverity := E_Severity.LOW,
            OperatorActionRequired := FALSE, LampTestRequest := FALSE,
            ParCfg := _towerCfg);
        IF TIME() - _towerStarted >= T#3MS THEN
            AssertFalse(Condition := _tower.Status.TestActive,
                Message := 'bounded test returns automatically to mapped state');
            _towerPhase := 0;
            TEST_FINISHED();
        ELSE
            ;
        END_IF
    ELSE
        _towerPhase := 0;
END_CASE
END_METHOD

METHOD Windows_clock_quality_rejects_bad_and_stale_samples
TEST('Windows_clock_quality_rejects_bad_and_stale_samples');
_clockSample.SchemaVersion := 1;
_clockSample.ByteCount := SIZEOF(_clockSample);
_clockSample.Magic := DWORD#16#434B5246;
_clockSample.Sequence := 1;
_clockSample.ObservedAt := DT#2026-10-06-00:00:00;
_clockSample.LastSyncAt := DT#2026-10-05-23:59:50;
_clockSample.OffsetUs := -25;
_clockSample.SyncAgeSeconds := 10;
_clockSample.ServiceError := 0;
_clockSample.Flags := DWORD#3;
_clockSample.Source := 'WINDOWS/W32TIME';
_clockSample.Crc := F_TcWindowsClockCrc(Sample := _clockSample);
_clockApplied := _windowsClock.M_ApplySample(Sample := _clockSample,
    WallNow := DT#2026-10-06-00:00:00, MonoNow := T#10S,
    MaximumSampleAge := T#90S, MaximumSyncAgeSeconds := 60, MaximumOffsetUs := 1000);
AssertTrue(Condition := _clockApplied AND _windowsClock.Quality.Synchronized,
    Message := 'fresh qualified Windows source is trusted');
AssertEquals_DINT(Expected := -25, Actual := _windowsClock.Quality.OffsetUs,
    Message := 'signed offset is preserved');

_clockApplied := _windowsClock.M_ApplySample(Sample := _clockSample,
    WallNow := DT#2026-10-06-00:01:31, MonoNow := T#101S,
    MaximumSampleAge := T#90S, MaximumSyncAgeSeconds := 60, MaximumOffsetUs := 1000);
AssertFalse(Condition := _windowsClock.Quality.Available,
    Message := 'observer expiry invalidates cached quality');

_clockSample.Sequence := 2;
_clockSample.OffsetUs := 1001;
_clockSample.Crc := F_TcWindowsClockCrc(Sample := _clockSample);
_clockApplied := _windowsClock.M_ApplySample(Sample := _clockSample,
    WallNow := DT#2026-10-06-00:00:00, MonoNow := T#102S,
    MaximumSampleAge := T#90S, MaximumSyncAgeSeconds := 60, MaximumOffsetUs := 1000);
AssertTrue(Condition := _windowsClock.Quality.Available,
    Message := 'excess offset is measured, not unavailable');
AssertFalse(Condition := _windowsClock.Quality.Synchronized,
    Message := 'excess offset cannot pass synchronization');

_clockSample.OffsetUs := 0;
_clockSample.ServiceError := 1062;
_clockSample.Flags := DWORD#0;
_clockSample.Crc := F_TcWindowsClockCrc(Sample := _clockSample);
_clockApplied := _windowsClock.M_ApplySample(Sample := _clockSample,
    WallNow := DT#2026-10-06-00:00:00, MonoNow := T#103S,
    MaximumSampleAge := T#90S, MaximumSyncAgeSeconds := 60, MaximumOffsetUs := 1000);
AssertFalse(Condition := _windowsClock.Quality.Available,
    Message := 'stopped Windows service is unavailable');

_clockSample.ServiceError := 0;
_clockSample.Flags := DWORD#3;
_clockSample.OffsetUs := 777;
// Deliberately omit recomputing the checksum: a corrupt record cannot pass.
_clockApplied := _windowsClock.M_ApplySample(Sample := _clockSample,
    WallNow := DT#2026-10-06-00:00:00, MonoNow := T#104S,
    MaximumSampleAge := T#90S, MaximumSyncAgeSeconds := 60, MaximumOffsetUs := 1000);
AssertFalse(Condition := _clockApplied OR _windowsClock.Quality.Synchronized,
    Message := 'corruption is fail-closed');
AssertEquals_DINT(Expected := 0, Actual := _windowsClock.Quality.OffsetUs,
    Message := 'a rejected record never publishes its bytes; the last accepted offset stands');

_clockSample.Crc := F_TcWindowsClockCrc(Sample := _clockSample);
_clockApplied := _windowsClock.M_ApplySample(Sample := _clockSample,
    WallNow := DT#2026-10-05-23:59:59, MonoNow := T#105S,
    MaximumSampleAge := T#90S, MaximumSyncAgeSeconds := 60, MaximumOffsetUs := 1000);
AssertTrue(Condition := _clockApplied AND _windowsClock.Quality.Synchronized,
    Message := 'a PLC clock a second behind the OS clock is within the record resolution');
_clockApplied := _windowsClock.M_ApplySample(Sample := _clockSample,
    WallNow := DT#2026-10-05-23:58:00, MonoNow := T#106S,
    MaximumSampleAge := T#90S, MaximumSyncAgeSeconds := 60, MaximumOffsetUs := 1000);
AssertTrue(Condition := _clockApplied AND _windowsClock.Quality.Available
    AND NOT _windowsClock.Quality.Synchronized,
    Message := 'a fresh record is still read, but a PLC clock minutes behind is not synchronized');
AssertEquals_UDINT(Expected := 1398, Actual := _windowsClock.ErrorID,
    Message := 'and says why: the PLC clock disagrees with the OS clock');
TEST_FINISHED();
END_METHOD

// One CRC for every wire record (F_Crc32), proven against the published check
// value and against a record the native x64 observer actually wrote on the test
// host (Windows Time stopped there: available=0, error 1062).
METHOD Crc32_matches_the_standard_and_the_native_observer
VAR
    check : ARRAY[0..8] OF BYTE := [49, 50, 51, 52, 53, 54, 55, 56, 57];
    native : ARRAY[0..75] OF BYTE := [
        1, 0, 76, 0, 70, 82, 75, 67, 228, 145, 137, 5, 113, 70, 197, 106, 0, 0, 0,
        0, 0, 0, 0, 0, 0, 0, 0, 0, 38, 4, 0, 0, 0, 0, 0, 0, 87, 73,
        78, 68, 79, 87, 83, 47, 87, 51, 50, 84, 73, 77, 69, 0, 0, 0, 0, 0, 0,
        0, 0, 0, 0, 0, 0, 0, 0, 0, 0, 0, 0, 0, 0, 0, 63, 189, 91, 179];
    sample : ST_TcWindowsClockSampleV1;
    reader : FB_TcWindowsTime;
END_VAR
TEST('Crc32_matches_the_standard_and_the_native_observer');
AssertEquals_DWORD(Expected := DWORD#16#CBF43926,
    Actual := F_Crc32(pData := ADR(check), Size := SIZEOF(check)),
    Message := 'the standard CRC-32 check value of 123456789');
AssertEquals_DWORD(Expected := 0, Actual := F_Crc32(pData := 0, Size := 4),
    Message := 'a null buffer is never read');
MEMCPY(destAddr := ADR(sample), srcAddr := ADR(native), n := SIZEOF(sample));
AssertEquals_DWORD(Expected := DWORD#16#B35BBD3F, Actual := F_TcWindowsClockCrc(Sample := sample),
    Message := 'the PLC computes the checksum the native observer wrote');
AssertTrue(Condition := reader.M_ApplySample(Sample := sample, WallNow := sample.ObservedAt,
    MonoNow := T#1S, MaximumSampleAge := T#90S, MaximumSyncAgeSeconds := 7200,
    MaximumOffsetUs := 1000), Message := 'a real observer record decodes in the PLC');
AssertFalse(Condition := reader.Quality.Available,
    Message := 'the stopped Windows Time service it recorded is unavailable quality');
AssertEquals_UDINT(Expected := 1062, Actual := reader.ErrorID,
    Message := 'with the service error the observer reported');
AssertEquals_STRING(Expected := 'WINDOWS/W32TIME', Actual := reader.Quality.Source,
    Message := 'and the source it named');
TEST_FINISHED();
END_METHOD

// The PLC file-reader path end to end through the real TwinCAT file service: a
// fresh record is read, a corrupted one is rejected, a missing file and a record
// that stops changing expire, a new record recovers - all without a PLC reset -
// and an event stamped meanwhile carries exactly the reader's synchronized flag.
METHOD Windows_clock_file_reader_reads_rejects_and_expires
VAR
    saved : ST_TimeQuality;
    slot : INT;
END_VAR
TEST('Windows_clock_file_reader_reads_rejects_and_expires');
_fileGuard(IN := _fileStep < 99, PT := T#40S);
IF _fileGuard.Q AND (_fileStep < 99) THEN
    AssertTrue(Condition := FALSE, Message := CONCAT(CONCAT(CONCAT('timed out in step ',
        INT_TO_STRING(_fileStep)), CONCAT(' reader error ', UDINT_TO_STRING(_fileClock.ErrorID))),
        CONCAT(' file error ', UDINT_TO_STRING(_fileOps.ErrorId))));
    _fileStep := 99;
    TEST_FINISHED();
    RETURN;
END_IF
_fileOps.Cyclic();
IF (_fileStep >= 3) AND (_fileStep < 99) THEN
    _fileClock.Cyclic(FilePath := CLOCK_TEST_FILE, PollInterval := T#1S,
        MaximumSampleAge := T#3S, MaximumSyncAgeSeconds := 7200, MaximumOffsetUs := 1000);
END_IF
CASE _fileStep OF
    0:
        IF _fileOps.M_MakeDir(Path := 'C:\ProgramData\Fraktal', Where := Tc2_System.PATH_GENERIC) THEN
            _fileStep := 1;         // an existing directory is not an error here
        END_IF
    1:
        IF NOT _fileOps.Busy AND _fileOps.M_MakeDir(Path := CLOCK_TEST_DIR, Where := Tc2_System.PATH_GENERIC) THEN
            _fileStep := 2;
        END_IF
    2:
        IF NOT _fileOps.Busy THEN
            _M_WriteClockSample(Sequence := 1, OffsetUs := 12, Corrupt := FALSE);
            _fileStep := 3;
        END_IF
    3:
        IF NOT _fileOps.Busy THEN
            AssertFalse(Condition := _fileOps.Error, Message := 'the observer record was staged');
            _fileStep := 4;
        END_IF
    4:
        IF _fileClock.Quality.Synchronized THEN
            AssertEquals_DINT(Expected := 12, Actual := _fileClock.Quality.OffsetUs,
                Message := 'the reader publishes the measured offset');
            saved := GVL_FraktalTime.Current;
            GVL_FraktalTime.Current := _fileClock.Quality;
            slot := _fileLog.Raise(Reason := E_Reason.NONE, Text := 'test.synchronized',
                Source := 'Test.Clock', Severity := E_Severity.LOW,
                Category := E_Category.SYSTEM, ResetClass := E_ResetClass.AUTO_RESET);
            AssertTrue(Condition := _fileLog.Active[slot].ComeTimeSynchronized,
                Message := 'an event stamped from a synchronized reader says so');
            _fileLog.Gone(Slot := slot);
            GVL_FraktalTime.Current := saved;
            _M_WriteClockSample(Sequence := 2, OffsetUs := 12, Corrupt := TRUE);
            _fileStep := 5;
        END_IF
    5:
        IF NOT _fileOps.Busy AND NOT _fileClock.Quality.Available
            AND (_fileClock.ErrorID = 13) THEN
            saved := GVL_FraktalTime.Current;
            GVL_FraktalTime.Current := _fileClock.Quality;
            slot := _fileLog.Raise(Reason := E_Reason.NONE, Text := 'test.unavailable',
                Source := 'Test.Clock', Severity := E_Severity.LOW,
                Category := E_Category.SYSTEM, ResetClass := E_ResetClass.AUTO_RESET);
            AssertFalse(Condition := _fileLog.Active[slot].ComeTimeSynchronized,
                Message := 'an event stamped while the record is corrupt is not synchronized');
            _fileLog.Gone(Slot := slot);
            GVL_FraktalTime.Current := saved;
            _fileOps.M_Delete(Path := CLOCK_TEST_FILE, Where := Tc2_System.PATH_GENERIC);
            _fileStep := 6;
        END_IF
    6:
        IF NOT _fileOps.Busy THEN
            IF _fileOps.Error THEN
                // The reader holds the file for a few scans per poll, without
                // delete-sharing: a delete that met it is simply retried.
                _fileOps.M_Delete(Path := CLOCK_TEST_FILE, Where := Tc2_System.PATH_GENERIC);
            ELSIF _fileClock.ErrorID = 16#70C THEN
                AssertFalse(Condition := _fileClock.Quality.Available,
                    Message := 'a missing observer record is unavailable and says why (not found)');
                _M_WriteClockSample(Sequence := 3, OffsetUs := -40, Corrupt := FALSE);
                _fileStep := 7;
            END_IF
        END_IF
    7:
        IF NOT _fileOps.Busy AND _fileClock.Quality.Synchronized THEN
            AssertEquals_DINT(Expected := -40, Actual := _fileClock.Quality.OffsetUs,
                Message := 'a new record recovers without a PLC reset');
            _fileStep := 8;         // and is never rewritten again
        END_IF
    8:
        IF NOT _fileClock.Quality.Available THEN
            AssertEquals_UDINT(Expected := 1460, Actual := _fileClock.ErrorID,
                Message := 'a record that stops changing expires (stale observer)');
            _fileOps.M_Delete(Path := CLOCK_TEST_FILE, Where := Tc2_System.PATH_GENERIC);
            _fileStep := 9;
        END_IF
    9:
        IF NOT _fileOps.Busy THEN
            IF _fileOps.Error THEN
                _fileOps.M_Delete(Path := CLOCK_TEST_FILE, Where := Tc2_System.PATH_GENERIC);
            ELSE
                _fileStep := 99;
                TEST_FINISHED();
            END_IF
        END_IF
    99:
        ;
ELSE
    _fileStep := 99;
END_CASE
END_METHOD

// Stage a record exactly as the native observer writes it: synchronized just now.
METHOD PRIVATE _M_WriteClockSample : BOOL
VAR_INPUT
    Sequence : UDINT;
    OffsetUs : DINT;
    Corrupt : BOOL;
END_VAR
MEMSET(destAddr := ADR(_fileSample), fillByte := 0, n := SIZEOF(_fileSample));
_fileSample.SchemaVersion := 1;
_fileSample.ByteCount := TO_UINT(SIZEOF(_fileSample));
_fileSample.Magic := DWORD#16#434B5246;
_fileSample.Sequence := Sequence;
_fileSample.ObservedAt := F_Now();
_fileSample.LastSyncAt := _fileSample.ObservedAt;
_fileSample.OffsetUs := OffsetUs;
_fileSample.SyncAgeSeconds := 0;
_fileSample.ServiceError := 0;
_fileSample.Flags := DWORD#3;
_fileSample.Source := 'WINDOWS/W32TIME';
_fileSample.Crc := F_TcWindowsClockCrc(Sample := _fileSample);
IF Corrupt THEN
    _fileSample.Crc := _fileSample.Crc XOR DWORD#1;
END_IF
_M_WriteClockSample := _fileOps.M_Write(Path := CLOCK_TEST_FILE, Where := Tc2_System.PATH_GENERIC,
    pData := ADR(_fileSample), Size := SIZEOF(_fileSample));
END_METHOD

END_FUNCTION_BLOCK

// ---- Fraktal_Tests/FB_ProbeFileOps.TcPOU
// Test-only file operations on the isolated test runtime: delete a file, write
// raw bytes, create or remove a directory - the damage a power cut, an operator or
// a full disk does to retained data, staged deliberately. One operation at a time:
// start it with an M_ call while Busy is FALSE, then call Cyclic until Busy drops.
FUNCTION_BLOCK FB_ProbeFileOps
VAR_OUTPUT
    Busy    : BOOL;
    Error   : BOOL;     // the last operation failed
    ErrorId : UDINT;
END_VAR
VAR
    _delete : Tc2_System.FB_FileDelete;
    _mkdir  : Tc2_System.FB_CreateDir;
    _rmdir  : Tc2_System.FB_RemoveDir;
    _open   : Tc2_System.FB_FileOpen;
    _write  : Tc2_System.FB_FileWrite;
    _close  : Tc2_System.FB_FileClose;
    _phase  : INT;
    _path   : STRING(255);
    _where  : Tc2_System.E_OpenPath;
    _pData  : PVOID;
    _size   : UDINT;
    _handle : UINT;
END_VAR

;

METHOD M_Delete : BOOL
VAR_INPUT
    Path  : STRING(255);
    Where : Tc2_System.E_OpenPath;
END_VAR
M_Delete := _M_Start(Path := Path, Where := Where, Phase := 10);
END_METHOD

METHOD M_MakeDir : BOOL
VAR_INPUT
    Path  : STRING(255);
    Where : Tc2_System.E_OpenPath;
END_VAR
M_MakeDir := _M_Start(Path := Path, Where := Where, Phase := 20);
END_METHOD

METHOD M_RemoveDir : BOOL
VAR_INPUT
    Path  : STRING(255);
    Where : Tc2_System.E_OpenPath;
END_VAR
M_RemoveDir := _M_Start(Path := Path, Where := Where, Phase := 30);
END_METHOD

// Create or truncate Path and write Size bytes from pData.
METHOD M_Write : BOOL
VAR_INPUT
    Path  : STRING(255);
    Where : Tc2_System.E_OpenPath;
    pData : PVOID;
    Size  : UDINT;
END_VAR
_pData := pData;
_size := Size;
M_Write := _M_Start(Path := Path, Where := Where, Phase := 40);
END_METHOD

METHOD Cyclic : BOOL
CASE _phase OF
    0:
        ;
    10:
        _delete(bExecute := FALSE);
        _delete(sNetId := '', sPathName := _path, ePath := _where, bExecute := TRUE, tTimeout := T#3S);
        _phase := 11;
    11:
        _delete(bExecute := FALSE);
        IF NOT _delete.bBusy THEN
            _M_Done(Failed := _delete.bError, Id := _delete.nErrId);
        END_IF
    20:
        _mkdir(bExecute := FALSE);
        _mkdir(sNetId := '', sPathName := _path, ePath := _where, bExecute := TRUE, tTimeout := T#3S);
        _phase := 21;
    21:
        _mkdir(bExecute := FALSE);
        IF NOT _mkdir.bBusy THEN
            _M_Done(Failed := _mkdir.bError, Id := _mkdir.nErrId);
        END_IF
    30:
        _rmdir(bExecute := FALSE);
        _rmdir(sNetId := '', sPathName := _path, ePath := _where, bExecute := TRUE, tTimeout := T#3S);
        _phase := 31;
    31:
        _rmdir(bExecute := FALSE);
        IF NOT _rmdir.bBusy THEN
            _M_Done(Failed := _rmdir.bError, Id := _rmdir.nErrId);
        END_IF
    40:
        _open(bExecute := FALSE);
        _open(sNetId := '', sPathName := _path,
            nMode := Tc2_System.FOPEN_MODEWRITE OR Tc2_System.FOPEN_MODEBINARY,
            ePath := _where, bExecute := TRUE, tTimeout := T#3S);
        _phase := 41;
    41:
        _open(bExecute := FALSE);
        IF NOT _open.bBusy THEN
            IF _open.bError THEN
                _M_Done(Failed := TRUE, Id := _open.nErrId);
            ELSE
                _handle := _open.hFile;
                _write(bExecute := FALSE);
                _write(sNetId := '', hFile := _handle, pWriteBuff := _pData,
                    cbWriteLen := _size, bExecute := TRUE, tTimeout := T#3S);
                _phase := 42;
            END_IF
        END_IF
    42:
        _write(bExecute := FALSE);
        IF NOT _write.bBusy THEN
            Error := _write.bError OR (_write.cbWrite <> _size);
            ErrorId := _write.nErrId;
            _close(bExecute := FALSE);
            _close(sNetId := '', hFile := _handle, bExecute := TRUE, tTimeout := T#3S);
            _phase := 43;
        END_IF
    43:
        _close(bExecute := FALSE);
        IF NOT _close.bBusy THEN
            _M_Done(Failed := Error OR _close.bError, Id := SEL(_close.bError, ErrorId, _close.nErrId));
        END_IF
ELSE
    _M_Done(Failed := TRUE, Id := 0);
END_CASE
Cyclic := NOT Busy;
END_METHOD

METHOD PRIVATE _M_Start : BOOL
VAR_INPUT
    Path  : STRING(255);
    Where : Tc2_System.E_OpenPath;
    Phase : INT;
END_VAR
_M_Start := FALSE;
IF Busy THEN
    RETURN;
END_IF
_path := Path;
_where := Where;
_phase := Phase;
Busy := TRUE;
Error := FALSE;
ErrorId := 0;
_M_Start := TRUE;
END_METHOD

METHOD PRIVATE _M_Done
VAR_INPUT
    Failed : BOOL;
    Id     : UDINT;
END_VAR
Error := Failed;
ErrorId := Id;
Busy := FALSE;
_phase := 0;
END_METHOD

END_FUNCTION_BLOCK

// ---- Fraktal_Tests/FB_SequenceRaise_Tests.TcPOU
// Core §6.9 — an error raised BY a step, for the cases `Awaits` cannot reach:
// a command behind an IF, and a rule only the application knows. Proves the three
// promised behaviours: the chain stops, the §3.13 row carries the drill-down link,
// and clearing the error re-evaluates the command instead of resuming blind.
FUNCTION_BLOCK FB_SequenceRaise_Tests EXTENDS TcUnit.FB_TestSuite
VAR
    _u : FB_ProbeUnitRaise;
    _x : FB_ProbeUnitRaise;   // custom-message path, entered at step 30 cleanly
    _v : FB_ProbeUnitRaise;   // warning path, kept off the fault path's state
    _r : FB_ProbeUnitRaise;   // report-without-adopting path (press AUTO N200)
    _w1, _w2, _w3, _w4, _w5 : BOOL;
    _ringBefore : INT;
END_VAR

Guarded_child_fault_is_raised_with_its_drilldown_link();
Cleared_error_re_evaluates_the_command_at_the_same_step();
Custom_message_carries_its_own_severity_and_link();
Warning_is_recorded_once_per_visit_and_stops_nothing();
Reported_child_failure_is_visible_without_stopping_the_chain();

METHOD Guarded_child_fault_is_raised_with_its_drilldown_link
VAR
    d : ST_Diagnostic;
END_VAR
TEST('Guarded_child_fault_is_raised_with_its_drilldown_link');
IF NOT _w1 THEN
    AssertTrue(Condition := _u.Setup(Name := 'Test.Raise'), Message := 'Unit sets up');
    _u.Enable := TRUE;                   // the IF that hides the child from `Awaits`
    AssertTrue(Condition := _u.Start(), Message := 'Unit starts');
    _u();                                // edge -> BUSY; chain step 10 -> 20
    _u();                                // step 20 issues the guarded command
    AssertEquals_UDINT(Expected := 1, Actual := _u.M_TestIssues(),
        Message := 'the guarded command was issued once (§6.1 one-shot)');
    AssertFalse(Condition := _u.Error, Message := 'no fault while the child runs');
    _u.M_TestSetChild(ChildDone := FALSE, ChildFault := TRUE);
    _u();                                // children tick first, then the step raises
    AssertTrue(Condition := _u.Error,
        Message := 'a raised child fault stops the chain, exactly like an awaited one');
    d := _u.GetFaultSummary();
    AssertEquals_DWORD(Expected := TO_DWORD(E_Reason.TEST_FAULT),
        Actual := TO_DWORD(d.ReasonCode),
        Message := 'the child first-out is adopted verbatim, not re-invented');
    AssertEquals_STRING(Expected := 'Test.Raise.Child', Actual := d.SourcePath,
        Message := 'the failing module owns the diagnostic (§8.2)');
    AssertEquals_INT(Expected := 20, Actual := _u.M_TestChainStep(),
        Message := 'the chain stopped ON the step; a raise never advances it');
    AssertEquals_INT(Expected := 2, Actual := _u.SequenceStepCount,
        Message := 'the chart holds the steps reached so far - step 30 is honestly absent');
    AssertTrue(Condition := _u.SequenceSteps[2].ErrorActive,
        Message := 'the raising row is marked, so the chart can blink it red');
    AssertEquals_STRING(Expected := 'Test.Raise.Child',
        Actual := M_NotePath(Unit := _u, RowIdx := 2, IsError := TRUE),
        Message := 'the row is click-through to the module that failed, even though the step passed Awaits := 0');
    // One more cyclic pass WHILE the Unit is in ERROR. FB_UnitBase samples the
    // error-cleared edge inside OnCyclic, which runs BEFORE _M_Dispatch - so the
    // ERROR this scan's dispatch just raised is not visible to it yet, and if the
    // reset lands before any later scan the edge is never seen and the chain is
    // never re-armed. A real Unit sits in ERROR until an operator acts; a test
    // that resets in the same breath does not, and was measuring that instead.
    _u();
    AssertTrue(Condition := _u.Error, Message := 'still faulted before the reset');
    _w1 := TRUE;
END_IF
TEST_FINISHED();
END_METHOD

METHOD Cleared_error_re_evaluates_the_command_at_the_same_step
TEST('Cleared_error_re_evaluates_the_command_at_the_same_step');
IF NOT _w2 THEN
    _u.M_TestSetChild(ChildDone := TRUE, ChildFault := FALSE);   // cause removed
    AssertTrue(Condition := _u.OperatorReset(),
        Message := 'the reset releases the latched commands (§8.3(b))');
    _u();                                // Execute low -> READY: the ERROR-cleared edge
    AssertFalse(Condition := _u.SequenceSteps[2].ErrorActive,
        Message := 'the row error mark is cleared with the fault, not left stale');
    AssertTrue(Condition := _u.Start(), Message := 'restart after the reset');
    _u();                                // BUSY again; this project does not restart the chain
    AssertEquals_INT(Expected := 20, Actual := _u.M_TestChainStep(),
        Message := 'the chain resumes at the step that raised, not somewhere else');
    AssertEquals_UDINT(Expected := 2, Actual := _u.M_TestIssues(),
        Message := 're-evaluated: the command is issued again rather than assumed still running');
    // The child is already Done, so the re-issued command completes on the same
    // scan and the step advances once - a second call would run step 30 too.
    _u();                                // re-issued command completes -> step 30
    AssertEquals_INT(Expected := 30, Actual := _u.M_TestChainStep(),
        Message := 'the chain carries on once the step actually completes');
    _w2 := TRUE;
END_IF
TEST_FINISHED();
END_METHOD

METHOD Custom_message_carries_its_own_severity_and_link
VAR
    d : ST_Diagnostic;
END_VAR
TEST('Custom_message_carries_its_own_severity_and_link');
IF NOT _w3 THEN
    AssertTrue(Condition := _x.Setup(Name := 'Test.Raise'), Message := 'Unit sets up');
    _x.Enable := TRUE;
    _x.SimCustom := TRUE;                // the application rule step 30 checks
    _x.M_TestSetChild(ChildDone := TRUE, ChildFault := FALSE);
    AssertTrue(Condition := _x.Start(), Message := 'Unit starts');
    _x();                                // step 10 -> 20
    _x();                                // step 20 issues its command
    _x();                                // child Done -> step 30
    _x();                                // step 30 raises its own message
    AssertTrue(Condition := _x.Error, Message := 'a custom message stops the chain too');
    d := _x.GetFaultSummary();
    AssertEquals_STRING(Expected := 'project.test.customRaise', Actual := d.Description,
        Message := 'the step owns the text');
    AssertEquals_DWORD(Expected := TO_DWORD(E_Severity.HIGH), Actual := TO_DWORD(d.Severity),
        Message := 'an unregistered reason keeps the severity the step chose (§8.8)');
    AssertEquals_DWORD(Expected := TO_DWORD(E_Category.PROCESS), Actual := TO_DWORD(d.Category),
        Message := 'and the category it chose');
    AssertEquals_STRING(Expected := 'Test.Raise.Child', Actual := d.SourcePath,
        Message := 'a custom message may still point at the module that explains it');
    AssertTrue(Condition := _x.SequenceSteps[3].ErrorActive,
        Message := 'the custom raise marks its own §3.13 row');
    AssertEquals_STRING(Expected := 'Test.Raise.Child',
        Actual := M_NotePath(Unit := _x, RowIdx := 3, IsError := TRUE),
        Message := 'and publishes the link the chart drills into');
    _w3 := TRUE;
END_IF
TEST_FINISHED();
END_METHOD

METHOD Warning_is_recorded_once_per_visit_and_stops_nothing
TEST('Warning_is_recorded_once_per_visit_and_stops_nothing');
IF NOT _w4 THEN
    AssertTrue(Condition := _v.Setup(Name := 'Test.Warn'), Message := 'Unit sets up');
    _v.Enable := TRUE;
    _v.SimWarn := TRUE;
    // Hold the child OPEN so step 20 really is visited on two consecutive
    // scans - that is what the dedupe assertion below measures. With the
    // child pre-completed the step advanced on the scan it issued, so the
    // 'once per visit' claim was never actually exercised.
    _v.M_TestSetChild(ChildDone := FALSE, ChildFault := FALSE);
    AssertTrue(Condition := _v.Start(), Message := 'Unit starts');
    _v();                                // chain step 10 -> 20
    _ringBefore := _v.AlarmLog.RingHead;
    _v();                                // step 20: warning + the command
    _v();                                // still on step 20, called again every scan
    AssertFalse(Condition := _v.Error,
        Message := 'a warning is not a fault: the chain is never stopped by it');
    AssertTrue(Condition := _v.Busy, Message := 'and the Unit keeps running');
    AssertEquals_INT(Expected := (_ringBefore MOD PL_Fraktal.MAX_ALARM_RING) + 1,
        Actual := _v.AlarmLog.RingHead,
        Message := 'one ring entry per visit, not one per scan (§6.9(e) dedupe)');
    AssertEquals_DWORD(Expected := TO_DWORD(E_ResetClass.AUTO_RESET),
        Actual := TO_DWORD(_v.AlarmLog.Ring[_v.AlarmLog.RingHead].ResetClass),
        Message := 'AUTO_RESET come+gone: a message can never block the next Start');
    AssertFalse(Condition := _v.AlarmLog.Blocking,
        Message := 'and the log does not go blocking on it');
    AssertTrue(Condition := _v.SequenceSteps[2].WarningActive,
        Message := 'the §3.13 row carries the message');
    AssertEquals_STRING(Expected := 'project.test.stepWarning',
        Actual := M_NoteKey(Unit := _v, RowIdx := 2, IsError := FALSE),
        Message := 'with the key the step chose');
    _v.M_TestSetChild(ChildDone := TRUE, ChildFault := FALSE);
    _v();                                // child Done -> advance
    AssertEquals_INT(Expected := 30, Actual := _v.M_TestChainStep(),
        Message := 'the step completed normally: the warning changed no flow');
    _w4 := TRUE;
END_IF
TEST_FINISHED();
END_METHOD

METHOD Reported_child_failure_is_visible_without_stopping_the_chain
TEST('Reported_child_failure_is_visible_without_stopping_the_chain');
IF NOT _w5 THEN
    AssertTrue(Condition := _r.Setup(Name := 'Test.Report'), Message := 'Unit sets up');
    _r.Enable := TRUE;
    _r.ReportOnly := TRUE;               // the step owns the recovery, like press AUTO N200
    AssertTrue(Condition := _r.Start(), Message := 'Unit starts');
    _r();                                // step 10 -> 20
    _r();                                // step 20 issues the command
    _r.M_TestSetChild(ChildDone := FALSE, ChildFault := TRUE);
    _r();                                // the child fails; the step reports and routes
    AssertFalse(Condition := _r.Error,
        Message := 'reporting is not adopting: the Unit does not fault');
    AssertTrue(Condition := _r.Busy, Message := 'and the chain keeps running');
    AssertTrue(Condition := _r.SequenceSteps[2].WarningActive,
        Message := 'the failure is visible on the §3.13 row that handled it');
    AssertEquals_STRING(Expected := 'probe fault',
        Actual := M_NoteKey(Unit := _r, RowIdx := 2, IsError := FALSE),
        Message := 'with the CHILD text verbatim, not a re-invented one');
    AssertEquals_STRING(Expected := 'Test.Report.Child',
        Actual := M_NotePath(Unit := _r, RowIdx := 2, IsError := FALSE),
        Message := 'and click-through to the module that failed, with Awaits := 0');
    AssertFalse(Condition := _r.SequenceSteps[2].ErrorActive,
        Message := 'a reported failure never borrows the error mark');
    // The report and the ADVANCE happen in the SAME scan the child fails:
    // M_ReportFromChild does not RETURN, so M_Advance(OnAdvance := 30) runs
    // below it. An extra call here would run step 30 too and land on 999.
    AssertEquals_INT(Expected := 30, Actual := _r.M_TestChainStep(),
        Message := 'the chain took its own recovery branch instead of stopping');
    _w5 := TRUE;
END_IF
TEST_FINISHED();
END_METHOD

// Core §6.9 — the annotation attached to one §3.13 row, or 0 if it has none.
// The row keeps only the MARK; the key and the drill-down path are in the sparse
// annotation table, so a row stays correctly coloured even when that table is full.
METHOD M_NoteIdx : INT
VAR_INPUT
    Unit : REFERENCE TO FB_ProbeUnitRaise;
    RowIdx : INT;
    IsError : BOOL;
END_VAR
VAR
    i : INT;
END_VAR
FOR i := 1 TO Unit.SequenceAnnotationCount DO
    IF (Unit.SequenceAnnotations[i].RowIdx = RowIdx)
    AND (Unit.SequenceAnnotations[i].IsError = IsError) THEN
        M_NoteIdx := i;
        RETURN;
    END_IF
END_FOR
END_METHOD

// '' when the row has no such annotation, so a missing one fails the assertion
// with '' instead of indexing outside the table.
METHOD M_NoteKey : STRING(120)
VAR_INPUT
    Unit : REFERENCE TO FB_ProbeUnitRaise;
    RowIdx : INT;
    IsError : BOOL;
END_VAR
VAR
    idx : INT;
END_VAR
idx := M_NoteIdx(Unit := Unit, RowIdx := RowIdx, IsError := IsError);
IF idx > 0 THEN
    M_NoteKey := Unit.SequenceAnnotations[idx].Key;
END_IF
END_METHOD

METHOD M_NotePath : STRING(80)
VAR_INPUT
    Unit : REFERENCE TO FB_ProbeUnitRaise;
    RowIdx : INT;
    IsError : BOOL;
END_VAR
VAR
    idx : INT;
END_VAR
idx := M_NoteIdx(Unit := Unit, RowIdx := RowIdx, IsError := IsError);
IF idx > 0 THEN
    M_NotePath := Unit.SequenceAnnotations[idx].SourcePath;
END_IF
END_METHOD

END_FUNCTION_BLOCK

// ---- Fraktal_Tests/FB_ProbeUnitRaise.TcPOU
// Unit host for the §6.9 raise suite. Wiring only - every step lives in the chain.
// It registers its child but deliberately does NOT call _M_RollupFault: that is the
// whole scenario. A child commanded behind an IF cannot be handed to `Awaits`, so
// without an explicit raise its fault would leave the chain waiting until the stall
// guard, with nothing naming what broke.
FUNCTION_BLOCK FB_ProbeUnitRaise EXTENDS FB_UnitBase
VAR_INPUT
    Enable    : BOOL;
    SimCustom : BOOL;
    SimWarn   : BOOL;
    ReportOnly : BOOL;
    // Whether a fresh run command restarts the chain (the demo's choice) or lets it
    // resume where the error stopped it. Both are legitimate; the project decides.
    RestartOnCommand : BOOL;
END_VAR
VAR
    Child : FB_ProbeCM;
    Chain : FB_ProbeRaiseChain;
END_VAR

Cyclic();

METHOD Setup : BOOL
VAR_INPUT
    Name : STRING(80);
END_VAR
_M_SetName(Name);
StallTime := T#10S;                      // long: this suite tests raises, not stalls
Setup := Child.Setup(Name := CONCAT(Name, '.Child'))
    AND _M_Register(Child := Child)
    AND Chain.Setup(Host := THIS^, Child := Child);
END_METHOD

METHOD PROTECTED OnCyclic : DINT
OnCyclic := SUPER^.OnCyclic();   // base first (Core §3.14.2)
_M_TickChildren();
END_METHOD

METHOD PROTECTED _M_Dispatch
Chain.Enable := Enable;
Chain.SimCustom := SimCustom;
Chain.SimWarn := SimWarn;
Chain.ReportOnly := ReportOnly;
Chain.M_Run();
END_METHOD

METHOD PROTECTED OnCommandStart : DINT
OnCommandStart := SUPER^.OnCommandStart();
IF RestartOnCommand THEN
    Chain.M_Reset();
END_IF
END_METHOD

// Test injection stays inside the owning FB (see FB_ProbeEM).
METHOD M_TestSetChild : BOOL
VAR_INPUT
    ChildDone  : BOOL;
    ChildFault : BOOL;
END_VAR
Child.SimDone := ChildDone;
Child.SimFault := ChildFault;
M_TestSetChild := TRUE;
END_METHOD

// test seam: how many times the guarded command was actually issued
METHOD M_TestIssues : UDINT
M_TestIssues := Chain.Issues;
END_METHOD

// test seam: the chain's own active step, which a raise must not move
METHOD M_TestChainStep : INT
M_TestChainStep := Chain.ActiveStep;
END_METHOD

END_FUNCTION_BLOCK

// ---- Fraktal_Tests/FB_ProbeRaiseChain.TcPOU
// Core §6.9 — the worked example for an explicitly raised step error. Its two
// steps are the two shapes a chain cannot express with `Awaits`: a command
// guarded by an IF (so the framework never sees the child), and a rule only the
// application knows. Both stop the chain; both re-evaluate on resume.
FUNCTION_BLOCK FB_ProbeRaiseChain EXTENDS FB_SequenceBase
VAR_INPUT
    Enable    : BOOL;               // the IF that hides the child from `Awaits`
    SimCustom : BOOL;               // the application rule step 30 checks
    SimWarn   : BOOL;               // the non-blocking message step 20 reports
    ReportOnly : BOOL;              // step 20 owns the recovery, like press AUTO N200
END_VAR
VAR_OUTPUT
    Issues : UDINT;                 // times step 20 issued its command (§6.1 one-shot)
    Warned : BOOL;                  // last M_RaiseWarning result
    Reported : BOOL;                // last M_ReportFromChild result
END_VAR
VAR
    {attribute 'OPC.UA.DA' := '0'}
    _child : REFERENCE TO FB_ProbeCM;
END_VAR

;

METHOD Setup : BOOL
VAR_INPUT
    Host : I_SequenceHost;
END_VAR
VAR_IN_OUT
    Child : FB_ProbeCM;
END_VAR
_child REF= Child;
Setup := M_Attach(Host := Host) AND __ISVALIDREF(_child);
END_METHOD

METHOD M_Reset
M_ResetBase(FirstStep := 0);
Issues := 0;
Warned := FALSE;
Reported := FALSE;
END_METHOD

